	FOR nItemIndex :=1 TO cMAX_VALIDATION_ITEMS DO
		IF eCodeAIType = stCodeInfo.stGS1_Field[nItemIndex].eGS1_AIType THEN
			stItem := stCodeInfo.stGS1_Field[nItemIndex];
			EXIT;
		ELSE
			F_GS1_GetItem := 'Validation Item Not Found';
		END_IF
	END_FOR


	IF stItem.sStartAI <> '' AND stItem.sEndAI <> '' THEN
		nStart := FIND(sFullCode, stItem.sStartAI) + LEN(stItem.sStartAI);
		IF nStart > 0 THEN
			sTemp := RIGHT(sFullCode, LEN(sFullCode) - (nStart - 1));
		ELSE
			sTemp := sFullCode;
		END_IF
		nEnd := FIND(sTemp, stItem.sEndAI);
		IF nEnd = 0 THEN
			nEnd := LEN(sFullCode)+1;
		ELSE
			nEnd := nEnd +(nStart - 1);
		END_IF
	ELSIF stItem.sStartAI <> '' AND stItem.nCodeLength > 0 THEN
		nStart := FIND(sFullCode, stItem.sStartAI) + LEN(stItem.sStartAI);
		nEnd := nStart + stItem.nCodeLength;
	ELSIF stItem.nCodeStartPos > 0 AND stItem.sEndAI <> '' THEN
		nStart := stItem.nCodeStartPos;
		sTemp := RIGHT(sFullCode, LEN(sFullCode) - (nStart - 1));
		nEnd := FIND(sTemp, stItem.sEndAI);
		IF nEnd = 0 THEN
			nEnd := LEN(sFullCode)+1;
		ELSE
			nEnd := nEnd +(nStart - 1);
		END_IF
	ELSIF stItem.nCodeStartPos >= 0 AND stItem.nCodeLength > 0 THEN
		nStart := stItem.nCodeStartPos;
		nEnd := nStart + stItem.nCodeLength;
	ELSE
		nStart := 0;
		nEnd := 0;
	END_IF
	IF nStart > 0 AND nEnd > 0 THEN
		sItem := MID(sFullCode, nEnd - nStart, nStart);
	ELSE
		sItem := '';
	END_IF
ELSE
	sItem := '';
END_IF

F_GS1_GetItem := sItem;

END_FUNCTION

// ---- POUs/METS/Common LIB/08_SOFTWARE LIB/Cog Checker FB/FB_CogCorrection.TcPOU
FUNCTION_BLOCK FB_CogCorrection
VAR_INPUT
	bStart:		BOOL;
	bBailAfterFirstFound: BOOL;
	sSUPI:			STRING[12];
	nCorrectCogID:	INT;
END_VAR
VAR_OUTPUT
	bDone:			BOOL;
	sCorrectSUPI:	ARRAY[1..10] OF STRING[12];
END_VAR
VAR
	sModSUPI:	STRING[12];
	rtrigStart: R_TRIG;
	nChar: INT;
	nPos: INT;
	nStep: INT;
	sChar: STRING[1];
	DIGITS:				STRING[34] :=	'ABCDEFGHJKLMNPQRSTUVWXYZ0123456789';
	nCogResult: INT;
END_VAR

rtrigStart(CLK:= bStart);
IF rtrigStart.Q THEN
	nStep := 1;
END_IF

CASE nStep OF

	1:
		bDone := FALSE;
		MEMSET(ADR(sCorrectSUPI), 0, SIZEOF(sCorrectSUPI));

		sModSUPI := sSUPI;
		nChar := 1;
		nPos := 1;
		nStep := 2;

	2:
		FOR nChar := 1 TO 11 DO
						CheckResult();
			IF bDone THEN
				EXIT;
			END_IF
		END_FOR
		IF NOT(bDone) THEN
			nStep := 3;
		END_IF

	3:
		FOR nChar := 12 TO 23 DO
						CheckResult();
			IF bDone THEN
				EXIT;
			END_IF
		END_FOR
		IF NOT(bDone) THEN
			nStep := 4;
		END_IF


	4:
		FOR nChar := 24 TO 34 DO
						CheckResult();
			IF bDone THEN
				EXIT;
			END_IF
		END_FOR

		IF nPos < 12 THEN
			sModSUPI := sSUPI;
			nPos := nPos+1;
			nStep := 2;
		ELSE
			bDone := TRUE;
			nStep := 0;
		END_IF

END_CASE

ACTION CheckResult:
sChar := MID(DIGITS, 1, nChar);
sModSUPI := REPLACE(sModSUPI, sChar, 1, nPos);
nCogResult := F_COG_Checker(sModSUPI);
IF nCogResult = nCorrectCogID THEN
	MEMMOVE(ADR(sCorrectSUPI[2]), ADR(sCorrectSUPI[1]), SIZEOF(sCorrectSUPI) - SIZEOF(sCorrectSUPI[1]));
	sCorrectSUPI[1] := sModSUPI;
	IF bBailAfterFirstFound THEN
		bDone := TRUE;
		nStep := 0;
	END_IF
END_IF
END_ACTION

END_FUNCTION_BLOCK

// ---- POUs/METS/Common LIB/08_SOFTWARE LIB/Cog Checker FB/F_COG_Checker.TcPOU
FUNCTION F_COG_Checker : INT
VAR_INPUT
	sSUPI		: STRING[12];
END_VAR
VAR
	CogID		: INT;
	biCogID		: T_ULARGE_INTEGER;
	biLenDIGITS	: T_ULARGE_INTEGER;
	biPos		: T_ULARGE_INTEGER;
	biMSUPI_SIZE	: T_ULARGE_INTEGER;
	M			: T_ULARGE_INTEGER;
	biSUPI		: T_ULARGE_INTEGER;
	biPPrime		: T_ULARGE_INTEGER;
	biCODE_SIZE	: T_ULARGE_INTEGER;
	sM			: STRING[255];
	i			: INT;
	Pos			: DINT;
	strSUPI		: STRING[255];
END_VAR
VAR CONSTANT
	CODEGENID_SIZE	: DINT :=	49553;
	CODE_SIZE		: LREAL :=	2386420683693101056;
	DIGITS			: STRING[34] :=	'ABCDEFGHJKLMNPQRSTUVWXYZ0123456789';
	PPrime			: LREAL:= 618222249914457027;
END_VAR

	CogID := -1;
	biCODE_SIZE := LREAL_TO_UINT64(CODE_SIZE);
	biPPrime := LREAL_TO_UINT64(PPrime);

	(*MSUPI_SIZE := 10*366*24*60*1110*8232;*)
	biMSUPI_SIZE := STRING_TO_UINT64('48158385408000');

	bisupi := STRING_TO_UINT64('0');

	FOR i := LEN(sSUPI) TO 1 BY -1 DO
		Pos := FIND(DIGITS, MID(sSUPI, 1, i)) - 1;
		IF Pos >= 0 THEN
			(*supi := (supi* LEN(DIGITS)) + Pos;*)
			biPos.dwLowPart := TO_DWORD(Pos);
			biLenDIGITS.dwLowPart := TO_DWORD(LEN(DIGITS));
			biSUPI := UInt64Mul64(biSUPI, biLenDIGITS);
			biSUPI := UInt64Add64(biSUPI, biPos);
		END_IF
	END_FOR

	strSUPI := UINT64_TO_STRING(biSUPI);
	biPPrime := STRING_TO_UINT64('618222249914457027');
	biCODE_SIZE := STRING_TO_UINT64('2386420683693101056');

	M := F_MulMod(biPPrime, bisupi, biCODE_SIZE);
	sM := UINT64_TO_STRING(M);
	biCogID := UInt64Div64(M, biMSUPI_SIZE);
	CogID := DWORD_TO_INT(biCogID.dwLowPart);

IF CogID <= 0 OR CogID > CODEGENID_SIZE THEN
	CogID := -1;
END_IF

F_COG_Checker := CogID;

END_FUNCTION

// ---- POUs/METS/Common LIB/08_SOFTWARE LIB/Counter FBs/FB_ChangeStateTrig.TcPOU
FUNCTION_BLOCK FB_ChangeStateTrig
(*
Version history:
DATE		|	Version/Author 		|	Remark
----------------------------------------------------------------------------------------------------
16.03.12	|	2.000.001	PSA		|	Original Version.
									|	Monitors a boolean and gives a trigger on change of state
*)
VAR_INPUT
	bInput							: BOOL;			(* Variable to monitor *)
END_VAR
VAR_OUTPUT
	Q								: BOOL;			(* Output trigger *)
END_VAR
VAR
	bLastState						: BOOL;			(* Last known state of the variable *)
	fbTrig							: R_TRIG;		(* Trigger *)
END_VAR

fbTrig(CLK := bInput <> bLastState, Q => Q);
bLastState := bInput;

END_FUNCTION_BLOCK

// ---- POUs/METS/Common LIB/08_SOFTWARE LIB/Counter FBs/FB_CTD32.TcPOU
(* 32-bit counter with count value as VAR_IN_OUT to allow count value to be set externally *)
FUNCTION_BLOCK FB_CTD32
VAR_INPUT
	bInput			: BOOL;		(* FALSE-TRUE increments counter value *)
	bReset			: BOOL;		(* set TRUE to reset counter value to 0 *)
	nThreshold		: UDINT;	(* threshold at which bOutput is set TRUE *)
END_VAR
VAR_IN_OUT
	nCounter		: UDINT;	(* counter value *)
END_VAR
VAR_OUTPUT
	bOutput			: BOOL;		(* nCounter >= nTheshold *)
END_VAR
VAR
	fbInputEdge		: R_TRIG;
END_VAR
(*
-------------------------------------------------------------------------------------------------
Date		Version	Author	Comments
-------------------------------------------------------------------------------------------------
30/01/2015	3.00.00	PB		No change

-------------------------------------------------------------------------------------------------
05/02/10	1.00.00	PB		Initial release

-------------------------------------------------------------------------------------------------
*)

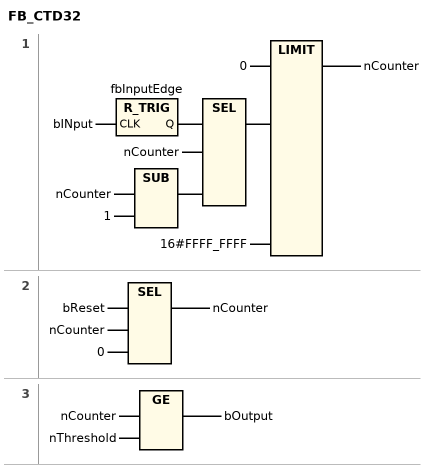
// NETWORK 1
fbInputEdge(CLK := bINput); // R_TRIG
nCounter := LIMIT(0, SEL(fbInputEdge.Q, nCounter, nCounter - 1), 16#FFFF_FFFF);

// NETWORK 2
nCounter := SEL(bReset, nCounter, 0);

// NETWORK 3
bOutput := nCounter >= nThreshold;

END_FUNCTION_BLOCK

// ---- POUs/METS/Common LIB/08_SOFTWARE LIB/Counter FBs/FB_CTU16.TcPOU
(* 16-bit counter with count value as VAR_IN_OUT to allow count value to be set externally *)
FUNCTION_BLOCK FB_CTU16
VAR_INPUT
	bInput			: BOOL;		(* FALSE-TRUE increments counter value *)
	bReset			: BOOL;		(* set TRUE to reset counter value to 0 *)
	nThreshold		: UINT;		(* threshold at which bOutput is set TRUE *)
END_VAR
VAR_IN_OUT
	nCounter		: UINT;		(* counter value *)
END_VAR
VAR_OUTPUT
	bOutput			: BOOL;		(* nCounter >= nTheshold *)
END_VAR
VAR
	fbInputEdge		: R_TRIG;
END_VAR
(*
-------------------------------------------------------------------------------------------------
Date		Version	Author	Comments
-------------------------------------------------------------------------------------------------
30/01/2015	3.00.00	PB		No change

-------------------------------------------------------------------------------------------------
05/02/10	1.00.00	PB		Initial release

-------------------------------------------------------------------------------------------------
*)

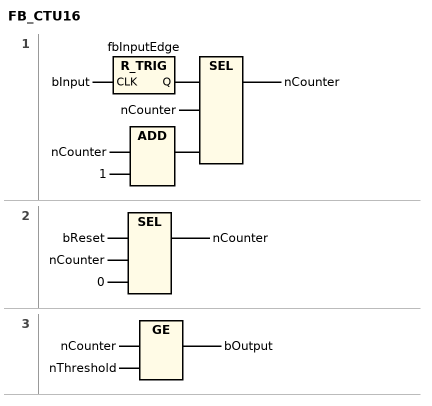
// NETWORK 1
fbInputEdge(CLK := bInput); // R_TRIG
nCounter := SEL(fbInputEdge.Q, nCounter, nCounter + 1);

// NETWORK 2
nCounter := SEL(bReset, nCounter, 0);

// NETWORK 3
bOutput := nCounter >= nThreshold;

END_FUNCTION_BLOCK

// ---- POUs/METS/Common LIB/08_SOFTWARE LIB/Counter FBs/FB_Incrementer.TcPOU
(* pulse incrementer with coarse and fine adjustment *)
FUNCTION_BLOCK FB_Incrementer
VAR_INPUT
	bIncrementHigh		: BOOL;		(* increment fValue in large steps *)
	bIncrementLow		: BOOL;		(* increment fValue in small steps *)
	bDecrementLow		: BOOL;		(* decrement fValue in small steps *)
	bDecrementHigh		: BOOL;		(* decrement fValue in large steps *)
	fLowIncValue		: LREAL;	(* large step change value *)
	fHighIncValue		: LREAL;	(* small step change value *)
END_VAR
VAR_IN_OUT
	fValue				: LREAL;	(* setpoint value *)
END_VAR
VAR
	fbIncrementHigh		: R_TRIG;
	fbIncrementLow		: R_TRIG;
	fbDecrementLow		: R_TRIG;
	fbDecrementHigh		: R_TRIG;
END_VAR
(*
-------------------------------------------------------------------------------------------------
Date		Version	Author	Comments
-------------------------------------------------------------------------------------------------
30/01/2015	3.00.00	PB		No change

-------------------------------------------------------------------------------------------------
26/09/2012	1.09.01	PB		Bug fix - output now LREAL instead of REAL
05/02/10	1.00.00	PB		Initial release

-------------------------------------------------------------------------------------------------
*)

(* add high increment value on rising edge of bIncrementHigh *)
fbIncrementHigh(CLK:= bIncrementHigh);
IF fbIncrementHigh.Q = TRUE THEN

	fValue := fValue + fHighIncValue;
END_IF

(* add low increment value on rising edge of bIncrementLow *)
fbIncrementLow(CLK:= bIncrementLow);
IF fbIncrementLow.Q = TRUE THEN

	fValue := fValue + fLowIncValue;
END_IF

(* subtract low increment value on rising edge of bDecrementLow *)
fbDecrementLow(CLK:= bDecrementLow);
IF fbDecrementLow.Q = TRUE THEN

	fValue := fValue - fLowIncValue;
END_IF

(* subtract high increment value on rising edge of bDecrementHigh *)
fbDecrementHigh(CLK:= bDecrementHigh);
IF fbDecrementHigh.Q = TRUE THEN

	fValue := fValue - fHighIncValue;
END_IF

END_FUNCTION_BLOCK

// ---- POUs/METS/Common LIB/08_SOFTWARE LIB/Counter FBs/FB_InWindow.TcPOU
(* set output when fActPos is within specified window, modulo roll-over is also accounted for *)
FUNCTION_BLOCK FB_InWindow
VAR_INPUT
	bEnable				: BOOL;		(* TRUE = enable output pulse *)
	fStartPos			: LREAL;	(* window start position *)
	fEndPos				: LREAL;	(* window end position *)
	fModuloFactor		: LREAL;	(* axis modulo factor, set to 0 for simple absolute window *)
	fActPos				: LREAL;	(* axis position *)
END_VAR
VAR_OUTPUT
	bInWindow			: BOOL;		(* TRUE = axis modulo position between fStartPos and fEndPos *)
	bStartWindow		: BOOL;		(* TRUE = one-shot pulse when axis has entered position window *)
	bEndWindow			: BOOL;		(* TRUE = one-shot pulse when axis has left position window *)
	fStartPosDiff		: LREAL;	(* pos diff between fStartPos and fActPos when bInWindow was set TRUE *)
END_VAR
VAR
	fbStartWindow		: R_TRIG;
	fbEndWindow			: F_TRIG;
	fCalcStartPos		: LREAL;
	fCalcEndPos			: LREAL;
	fCalcActPos			: LREAL;
END_VAR
(*
-------------------------------------------------------------------------------------------------
Date		Version	Author	Comments
-------------------------------------------------------------------------------------------------
30/01/2015	3.00.00	PB		No change

-------------------------------------------------------------------------------------------------
26/05/2011	1.06.04	PB		Can now set fModuloFactor to 0 to give simple absolute window detection
05/02/10	1.00.00	PB		Initial release

-------------------------------------------------------------------------------------------------

1.	If window is too small and fActPos passes fStartPos AND fEndPos in 1 PLC cycle, bInWindow will NOT be set.
2.	fActPos, fStartPos and fEndPos are automatically corrected for modulo positions, so input values can be
	outside of the modulo window without causing a problem.
*)

(* pulse output enabled *)
IF bEnable = TRUE THEN

	(* use modulo window *)
	IF fModuloFactor > 0 THEN

		(* apply modulo factor to fActPos, fStartPos and fEndPos *)
		fCalcActPos := LMOD(fActPos, fModuloFactor);
		fCalcStartPos := LMOD(fStartPos, fModuloFactor);
		fCalcEndPos := LMOD(fEndPos, fModuloFactor);
	
		(* pulse window does NOT cross modulo position boundary *)
		IF fCalcStartPos <= fCalcEndPos THEN
	
			(* axis modulo position is within defined window *)
			IF fCalcActPos >= fCalcStartPos AND fCalcActPos <= fCalcEndPos THEN
	
				(* set bInWindow output *)
				bInWindow := TRUE;
	
			(* axis modulo position is outside defined window *)
			ELSE
	
				(* reset bInWindow output *)
				bInWindow := FALSE;
			END_IF
	
		(* pulse window DOES cross modulo position boundary *)
		ELSE
	
			(* axis modulo position is within defined window *)
			IF (fCalcActPos >= fCalcStartPos AND fCalcActPos <= fModuloFactor) OR (fCalcActPos >= 0 AND fCalcActPos <= fCalcEndPos) THEN
	
				(* set bInWindow output *)
				bInWindow := TRUE;

			(* axis modulo position is outside defined window *)
			ELSE

				(* reset bInWindow output *)
				bInWindow := FALSE;
			END_IF
		END_IF

	(* use absolute window *)
	ELSE

		(* axis position is within defined window *)
		IF fActPos >= fStartPos AND fActPos <= fEndPos THEN

				(* set bInWindow output *)
			bInWindow := TRUE;

		(* axis position is outside defined window *)
		ELSE

				(* reset bInWindow output *)
			bInWindow := FALSE;
		END_IF
	END_IF


	(* give one-shot output pulse when axis enters defined window *)
	fbStartWindow(
		CLK := bInWindow,
		Q	=> bStartWindow
	);

	(* axis has entered position window *)
	IF bStartWindow = TRUE THEN

		(* calculate difference between target position and actual position when bInWindow is set TRUE *)
		fStartPosDiff := fCalcActPos - fCalcStartPos;
	END_IF

	(* give one-shot output pulse when axis leaves defined window *)
	fbEndWindow(
		CLK := bInWindow,
		Q	=> bEndWindow
	);

(* pulse output enabled *)
ELSE

	(* set outputs to 0, last start window pulse position is not affected *)
	bInWindow := FALSE;
	bStartWindow := FALSE;
	bEndWindow := FALSE;
END_IF

END_FUNCTION_BLOCK

// ---- POUs/METS/Common LIB/08_SOFTWARE LIB/File FBs/FB_FILE_ApendWriteByByte.TcPOU
(* write data from the source array to the target file in byte form *)
FUNCTION_BLOCK FB_FILE_ApendWriteByByte
VAR_INPUT
	bExecute			: BOOL;			(* set TRUE to write file *)
	pSourceAddr			: POINTER TO BYTE;	(* pointer to array of bytes containing data to be written *)
	nSourceSize			: UDINT;		(* number of bytes to write to file *)
	strPathFile			: T_MaxString;	(* path to file to be written *)
	tTimeout			: TIME;			(* timeout *)
END_VAR
VAR_OUTPUT
	bDone				: BOOL;			(* TRUE = file write complete *)
	bBusy				: BOOL;			(* TRUE = file write in progress *)
	bError				: BOOL;			(* TRUE = file write error *)
	nErrorID			: UDINT;		(* error code *)
	nBytesWritten		: UDINT;		(* bytes written to file *)
END_VAR
VAR
	eState				: E_FILE_State;
	eErrorState			: E_FILE_State;
	fbExecute			: R_TRIG;
	pWriteBuffer		: PVOID;
	nWriteBytes			: UDINT;
	fbOpenFile			: FB_FileOpen;
	hTarget				: UINT;
	fbWriteFile			: FB_FileWrite;
	fbCloseFile			: FB_FileClose;
	fbDelay				: TON;
END_VAR
(*
-------------------------------------------------------------------------------------------------
Date		Version	Author	Comments
-------------------------------------------------------------------------------------------------
03/11/2015	3.02.01	PB		Delay after FB_FileClose reduced from 10ms to 2ms
12/08/2015	3.02.00	PB		10ms delay added after FB_FileClose to ensure file has been released by OS before bDone is set TRUE
30/04/2015	3.00.00	PB		Moved from Sewtec_CaseTrace.lib
							Unknown state handling added

-------------------------------------------------------------------------------------------------
21/03/2012	1.37.04	PB		Number of bytes written by FB_FileWrite now checked against nSourceSize, re-write file if valus is incorrect
							Attempt to write file 3 times before returning error
02/03/2010	1.00.00	PB		Initial release

-------------------------------------------------------------------------------------------------
*)

(* rising edge of bExecute *)
fbExecute(CLK := bExecute);

CASE eState OF

	(* idle state *)
	E_FILE_IDLE:

		(* write data to binary file *)
		IF fbExecute.Q = TRUE THEN

			(* reset outputs *)
			bDone := FALSE;
			bBusy := TRUE;
			bError := FALSE;
			nErrorID := 0;
			nBytesWritten := 0;

			(* initialise vars *)
			eErrorState := eState;
			hTarget := 0;
			pWriteBuffer := pSourceAddr;
			nWriteBytes := nSourceSize;

			eState := E_FILE_OPEN;

		(* bExecute has been reset *)
		ELSIF bExecute = FALSE THEN

			bDone := FALSE;
			bBusy := FALSE;
			bError := FALSE;
			nErrorID := 0;

		END_IF


	(* open file *)
	E_FILE_OPEN:

		(* open file for writing in binary mode *)
		fbOpenFile(
			sNetId		:= '',
			sPathName	:= strPathFile,
			nMode		:= FOPEN_MODEAPPEND OR FOPEN_MODEPLUS OR FOPEN_MODEBINARY,
			ePath		:= PATH_GENERIC,
			bExecute	:= TRUE,
			tTimeout	:= tTimeout
		);

		(* file open completed *)
		IF fbOpenFile.bBusy = FALSE THEN

			(* file open completed OK *)
			IF fbOpenFile.bError = FALSE THEN

				(* log file handle for use by subsequent commands *)
				hTarget := fbOpenFile.hFile;

				eState := E_FILE_WRITE;

			(* file open error *)
			ELSE

				(* log error code and failure state *)
				bError := TRUE;
				nErrorID := fbOpenFile.nErrId;
				eErrorState := eState;

				(* abandon attempt to read file *)
				eState := E_FILE_DONE;
			END_IF

			(* close off fbOpenFile *)
			fbOpenFile(bExecute := FALSE);
		END_IF


	(* write file *)
	E_FILE_WRITE:

		(* write data to open file *)
		fbWriteFile(
			sNetId		:= '',
			hFile		:= hTarget,
			pWriteBuff	:= pWriteBuffer,
			cbWriteLen	:= nWriteBytes,
			bExecute	:= TRUE,
			tTimeout	:= tTimeout
		);

		(* file write completed *)
		IF fbWriteFile.bBusy = FALSE THEN

			(* file write completed OK *)
			IF fbWriteFile.bError = FALSE THEN

				(* log total bytes written *)
				nBytesWritten := fbWriteFile.cbWrite;

				eState := E_FILE_CLOSE;

			(* file write error *)
			ELSE

				(* no previous error *)
				IF bError = FALSE THEN

					(* log error code and failure state *)
					bError := TRUE;
					nErrorID := fbWriteFile.nErrId;
					eErrorState := eState;
				END_IF

				eState := E_FILE_CLOSE;
			END_IF

			(* close off fbReadFile *)
			fbWriteFile(bExecute := FALSE);
		END_IF


	(* close file *)
	E_FILE_CLOSE:

		(* close and release file for future use *)
		fbCloseFile(
			sNetId		:= '',
			hFile		:= hTarget,
			bExecute	:= TRUE,
			tTimeout	:= tTimeout,
		);

		(* file close completed *)
		IF fbCloseFile.bBusy = FALSE THEN

			(* file close completed OK *)
			IF fbCloseFile.bError = FALSE THEN

				eState := E_FILE_DONE;

			(* file close error *)
			ELSE

				(* no previous error *)
				IF bError = FALSE THEN

					(* log error code and failure state *)
					bError := TRUE;
					nErrorID := fbCloseFile.nErrId;
					eErrorState := eState;
				END_IF

				eState := E_FILE_DONE;
			END_IF

			(* reset delay timer *)
			fbDelay(IN := FALSE);

			(* close off fbCloseFile *)
			fbCloseFile(bExecute := FALSE);
		END_IF


	(* file access complete *)
	E_FILE_DONE:

		(* file close delay elapsed *)
		IF fbDelay.Q = TRUE THEN

			bDone := TRUE;
			bBusy := FALSE;
	
			eState := E_FILE_IDLE;
		END_IF


(* unknown state*)
ELSE

	eState := E_FILE_IDLE;

	(* update outputs *)
	bDone := TRUE;
	bBusy := FALSE;
	bError := TRUE;
	nErrorID := 16#FFFFFFFF;
	nBytesWritten := 0;
END_CASE

(* delay timer *)
fbDelay(
	IN	:= TRUE,
	PT	:= T#2ms
);

END_FUNCTION_BLOCK

// ---- POUs/METS/Common LIB/08_SOFTWARE LIB/File FBs/FB_FILE_Compare.TcPOU
(* read the attributes of 2 specified files and compare the file sizes in bytes *)
FUNCTION_BLOCK FB_FILE_Compare
VAR_INPUT
	bExecute			: BOOL;			(* set TRUE to compare specified files *)
	strPathFile1		: T_MaxString;	(* full path\file of 1st file for compare *)
	strPathFile2		: T_MaxString;	(* full path\file of 2nd file for compare *)
	tTimeout			: TIME;			(* timeout for each file operation *)
END_VAR
VAR_OUTPUT
	bDone				: BOOL;			(* TRUE = file access complete *)
	bBusy				: BOOL;			(* TRUE = file access in progress *)
	bError				: BOOL;			(* TRUE = error occurred during process *)
	nErrorID			: UDINT;		(* error code *)
	bFileMatchOK		: BOOL;			(* TRUE = files attributes match, valid when bDone = TRUE *)
END_VAR
VAR
	fbExecute			: R_TRIG;
	eState				: E_FILE_State;
	fbReadFileAttrib	: FB_EnumFindFileEntry;
	sFile1Attrib		: ST_FindFileEntry;
	sFile2Attrib		: ST_FindFileEntry;
	eErrorState			: E_FILE_State;
END_VAR
(*
-------------------------------------------------------------------------------------------------
Date		Version	Author	Comments
-------------------------------------------------------------------------------------------------
30/01/2015	3.00.00	PB		Moved from Sewtec_CaseTrace.lib

-------------------------------------------------------------------------------------------------
02/03/2010	1.00.00	PB		Initial release

-------------------------------------------------------------------------------------------------
*)

(* compare files on rising edge of bExecute *)
fbExecute(CLK := bExecute);

CASE eState OF

	(* initialise before scan *)
	E_FILE_IDLE:

		(* start new cycle *)
		IF fbExecute.Q = TRUE THEN

			(* reset outputs *)
			bDone := FALSE;
			bBusy := TRUE;
			bError := FALSE;
			nErrorID := 0;
			eErrorState := eState;
			bFileMatchOK := FALSE;

			eState := E_FILE_READ;

		(* reset status outputs when no cycle is required and bExecute is reset *)
		ELSIF bExecute = FALSE THEN

			bDone := FALSE;
			bBusy := FALSE;
			bError := FALSE;
			nErrorID := 0;
		END_IF


	(* read file 1 *)
	E_FILE_READ:

		(* read file attributes of file 1 *)
		fbReadFileAttrib(
			sNetId		:= '',
			sPathName	:= strPathFile1,
			eCmd		:= eEnumCmd_First,
			bExecute	:= TRUE,
			tTimeout	:= tTimeout,
			stFindFile	=> sFile1Attrib
		);

		(* file attribute read completed *)
		IF fbReadFileAttrib.bBusy = FALSE THEN

			(* file attributes read completed OK *)
			IF fbReadFileAttrib.bError = FALSE THEN

				(* end of entries not found, file exists *)
				IF fbReadFileAttrib.bEOE = FALSE THEN

					(* move to read attributes of File 2 *)
					eState := E_FILE_READ2;

				(* end of entries found, file does not exist *)
				ELSE

					(* no previous error *)
					IF bError = FALSE THEN
	
						bError := TRUE;
						nErrorID := 1;
						eErrorState := eState;
					END_IF

					(* resources held by fbReadFileAttrib released automatically *)
					eState := E_FILE_DONE;
				END_IF

			(* file read error *)
			ELSE

				(* log error code and failure state *)
				bError := TRUE;
				nErrorID := fbReadFileAttrib.nErrID;
				eErrorState := eState;

				(* end of entries found *)
				IF fbReadFileAttrib.bEOE = TRUE THEN

					(* resources released automatically by fbReadFileAttrib, move to compare file details *)
					eState := E_FILE_COMPARE;

				(* end of entries not found *)
				ELSE

					(* release resources held by fbReadFileAttrib *)
					eState := E_FILE_ABORT;
				END_IF
			END_IF

			(* close off fbReadFile *)
			fbReadFileAttrib(bExecute := FALSE);
		END_IF


	(* read file 2 *)
	E_FILE_READ2:

		(* read file attributes of file 2 *)
		fbReadFileAttrib(
			sNetId		:= '',
			sPathName	:= strPathFile2,
			eCmd		:= eEnumCmd_First,
			bExecute	:= TRUE,
			tTimeout	:= tTimeout,
			stFindFile	=> sFile2Attrib
		);

		(* file attribute read completed *)
		IF fbReadFileAttrib.bBusy = FALSE THEN

			(* file attributes read completed OK *)
			IF fbReadFileAttrib.bError = FALSE THEN

				(* end of entries not found, file exists *)
				IF fbReadFileAttrib.bEOE = FALSE THEN

					(* abort fbReadFileAttrib to release resources *)
					eState := E_FILE_ABORT;

				(* end of entries found, file does not exist *)
				ELSE

					(* no previous error *)
					IF bError = FALSE THEN
	
						bError := TRUE;
						nErrorID := 2;
						eErrorState := eState;
					END_IF

					(* resources held by fbReadFileAttrib released automatically *)
					eState := E_FILE_DONE;
				END_IF

			(* file read error *)
			ELSE

				(* log error code and failure state *)
				bError := TRUE;
				nErrorID := fbReadFileAttrib.nErrID;
				eErrorState := eState;

				(* end of entries found *)
				IF fbReadFileAttrib.bEOE = TRUE THEN

					(* resources released automatically by fbReadFileAttrib, move to compare file details *)
					eState := E_FILE_COMPARE;

				(* end of entries not found *)
				ELSE

					(* release resources held by fbReadFileAttrib *)
					eState := E_FILE_ABORT;
				END_IF
			END_IF

			(* close off fbReadFile *)
			fbReadFileAttrib(bExecute := FALSE);
		END_IF


	(* abort fbReadFileAttrib to release all resources *)
	E_FILE_ABORT:

		(* abort fbReadFileAttrib to release internal resources *)
		fbReadFileAttrib(
			eCmd		:= eEnumCmd_Abort,
			bExecute	:= TRUE,
		);

		(* abort file attricute read complete *)
		IF fbReadFileAttrib.bBusy = FALSE THEN

			(* abort file attricute read completed OK *)
			IF fbReadFileAttrib.bError = FALSE THEN

				(* no error occurred during file attribute read sequences *)
				IF bError = FALSE THEN

					(* move to COMPARE file attributes state *)
					eState := E_FILE_COMPARE;

				(* error occurred during file attribute read sequences *)
				ELSE

					(* move to COMPARE file attributes state *)
					eState := E_FILE_DONE;
				END_IF

			(* abort error *)
			ELSE

				(* no error occurred in previous states *)
				IF bError = FALSE THEN

					(* log error code and failure state *)
					bError := TRUE;
					nErrorID := fbReadFileAttrib.nErrID;
					eErrorState := eState;
				END_IF

				eState := E_FILE_DONE;
			END_IF

			(* close off fbReadFileAttrib *)
			fbReadFileAttrib(bExecute := FALSE);
		END_IF


	(* compare file attributes *)
	E_FILE_COMPARE:

		(* check if file size values (high and low dwords) are equal *)
		IF sFile1Attrib.fileSize.dwLowPart = sFile2Attrib.fileSize.dwLowPart
			AND sFile1Attrib.fileSize.dwHighPart = sFile2Attrib.fileSize.dwHighPart THEN

			bFileMatchOK := TRUE;	(* file sizes identical *)
		END_IF

		(* compare done *)
		eState := E_FILE_DONE;


	(* file access complete *)
	E_FILE_DONE:

		bDone := TRUE;
		bBusy := FALSE;

		(* return to IDLE state *)
		eState := E_FILE_IDLE;
END_CASE

END_FUNCTION_BLOCK

// ---- POUs/METS/Common LIB/08_SOFTWARE LIB/File FBs/FB_FILE_Copy.TcPOU
(* copy file(s) from SOURCE folder to TARGET folder, wildcard chars '*' and '?' can be used *)
FUNCTION_BLOCK FB_FILE_Copy
VAR_INPUT
	bExecute			: BOOL;			(* set TRUE to copy multiple files *)
	strPathSource		: T_MaxString;	(* folder path for SOURCE file*)
	strPathTarget		: T_MaxString;	(* folder path for TARGET file *)
	strFileName			: T_MaxString;	(* name of file to be copied *)
	tTimeout			: TIME;			(* timeout for each file operation *)
END_VAR
VAR_OUTPUT
	bDone				: BOOL;			(* TRUE = file access complete *)
	bBusy				: BOOL;			(* TRUE = file access in progress *)
	bError				: BOOL;			(* TRUE = error occurred during process *)
	nErrorID			: UDINT;		(* error code *)
	strOutputFile		: T_MaxString;	(* name of file that failed *)
END_VAR
VAR
	fbExecute			: R_TRIG;
	eState				: E_FILE_State;
	eErrorState			: E_FILE_State;
	fbFindFile			: FB_EnumFindFileEntry;
	eCommand			: E_EnumCmdType;
	strFoundFile		: T_MaxString;
	fbCopyFile			: FB_FILE_CopyByByte;
END_VAR
(*
-------------------------------------------------------------------------------------------------
Date		Version	Author	Comments
-------------------------------------------------------------------------------------------------
30/01/2015	3.00.00	PB		Moved from Sewtec_CaseTrace.lib

-------------------------------------------------------------------------------------------------
27/09/2010	1.05.03	PB		If a file cannot be copied, FB will now continue to next file in list rather than just abort and report an error
							strOutputFile will contain the name of the last file that failed
22/03/2010	1.02.00	PB		Initial release

-------------------------------------------------------------------------------------------------
*)

(* compare files on rising edge of bExecute *)
fbExecute(CLK := bExecute);

CASE eState OF

	(* idle state *)
	E_FILE_IDLE:

		(* start new cycle *)
		IF fbExecute.Q = TRUE THEN

			(* reset outputs *)
			bDone := FALSE;
			bBusy := TRUE;
			bError := FALSE;
			nErrorID := 0;
			strOutputFile := '';
			eErrorState := eState;

			eCommand := eEnumCmd_First;

			eState := E_FILE_FINDFILE;

		(* reset status outputs when no cycle is required and bExecute is reset *)
		ELSIF bExecute = FALSE THEN

			bDone := FALSE;
			bBusy := FALSE;
			bError := FALSE;
			nErrorID := 0;
			strOutputFile := '';
		END_IF


	(* find file *)
	E_FILE_FINDFILE:

		(* get file name *)
		fbFindFile(
			sNetId		:= '',
			sPathName	:= CONCAT(strPathSource, strFileName),
			eCmd		:= eCommand,
			bExecute	:= TRUE,
			tTimeout	:= T#1s,
		);

		(* get file name complete *)
		IF fbFindFile.bBusy = FALSE THEN

			(* get file name completed OK *)
			IF fbFindFile.bError = FALSE THEN

				(* file found *)
				IF fbFindFile.bEOE = FALSE THEN

					eCommand := eEnumCmd_Next;

					(* ignore filenames '.' and '..' *)
					IF fbFindFile.stFindFile.sFileName <> '.' AND fbFindFile.stFindFile.sFileName <> '..' THEN

						strFoundFile := fbFindFile.stFindFile.sFileName;
						eState := E_FILE_COPY;
					END_IF

				(* end of file list *)
				ELSE

					(* copy files complete *)
					eState := E_FILE_DONE;
				END_IF

			(* get file name error *)
			ELSE

				(* no error has previously occurred *)
				IF bError = FALSE THEN

					(* log error code and failure state *)
					bError := TRUE;
					nErrorID := fbFindFile.nErrId;
					eErrorState := eState;
				END_IF

				(* abandon attempt to copy files *)
				eState := E_FILE_ABORT;
			END_IF

			(* close off fbFindFile *)
			fbFindFile(bExecute := FALSE);
		END_IF


	(* copy file to TARGET folder *)
	E_FILE_COPY:

		(* copy files *)
		fbCopyFile(
			bExecute		:= TRUE,
			strPathSource	:= strPathSource,
			strPathTarget	:= strPathTarget,
			strFileName		:= strFoundFile,
			tTimeout		:= tTimeout,
		);

		(* copy file complete *)
		IF fbCopyFile.bDone = TRUE THEN

			(* copy file completed OK *)
			IF fbCopyFile.bError = FALSE THEN

				eState := E_FILE_FINDFILE;

			(* copy file error *)
			ELSE

				(* no error has previously occurred *)
				IF bError = FALSE THEN

					(* log error code and failure state *)
					strOutputFile := CONCAT(strPathSource, strFoundFile);
					bError := TRUE;
					nErrorID := fbCopyFile.nErrorID;
					eErrorState := eState;
				END_IF

				eState := E_FILE_FINDFILE;
			END_IF

			(* close off fbCopyFile *)
			fbCopyFile(bExecute := FALSE);
		END_IF


	(* abort file entry list *)
	E_FILE_ABORT:

		(* abort file entry list *)
		fbFindFile(
			sNetId		:= '',
			sPathName	:= '',
			eCmd		:= eEnumCmd_Abort,
			bExecute	:= TRUE,
			tTimeout	:= T#1s,
		);

		(* abort file entry complete *)
		IF fbFindFile.bBusy = FALSE THEN

			(* abort file entry completed OK *)
			IF fbFindFile.bError = FALSE THEN

				eState := E_FILE_DONE;

			(* abort file entry error *)
			ELSE

				(* no error has previously occurred *)
				IF bError = FALSE THEN

					(* log error code and failure state *)
					bError := TRUE;
					nErrorID := fbFindFile.nErrId;
					eErrorState := eState;
				END_IF

				(* abandon attempt to copy files *)
				eState := E_FILE_DONE;
			END_IF

			(* close off fbFindFile *)
			fbFindFile(bExecute := FALSE);
		END_IF


	(* file access complete *)
	E_FILE_DONE:

		bDone := TRUE;
		bBusy := FALSE;

		(* return to IDLE state *)
		eState := E_FILE_IDLE;

END_CASE

END_FUNCTION_BLOCK

// ---- POUs/METS/Common LIB/08_SOFTWARE LIB/File FBs/FB_FILE_CopyByByte.TcPOU
(* copy file from SOURCE to TARGET and verify, wildcard chars NOT allowed *)
FUNCTION_BLOCK FB_FILE_CopyByByte
VAR_INPUT
	bExecute			: BOOL;			(* set TRUE to copy file *)
	strPathSource		: T_MaxString;	(* folder path for SOURCE file*)
	strPathTarget		: T_MaxString;	(* folder path for TARGET file *)
	strFileName			: T_MaxString;	(* name of file to be copied*)
	tTimeout			: TIME;			(* timeout for each file operation *)
END_VAR
VAR_OUTPUT
	bDone				: BOOL;			(* TRUE = file access complete *)
	bBusy				: BOOL;			(* TRUE = file access in progress *)
	bError				: BOOL;			(* TRUE = error occurred during process *)
	nErrorID			: UDINT;		(* error code *)
END_VAR
VAR
	fbExecute			: R_TRIG;
	eState				: E_FILE_State;
	eErrorState			: E_FILE_State;
	fbGetFileSize		: FB_FILE_GetFileInfo;
	bFileSizeNotZero	: BOOL;
	fbOpenFile			: FB_FileOpen;
	hFileHandleSource	: UINT;
	hFileHandleTarget	: UINT;
	fbReadFile			: FB_FileRead;
	arrFileBytes		: ARRAY[0..32767] OF BYTE;
	nBytesRead			: UDINT;
	fbWriteFile			: FB_FileWrite;
	fbCloseFile			: FB_FileClose;
	fbFileCompare		: FB_FILE_Compare;
	bEOF				: BOOL;
END_VAR
(*
-------------------------------------------------------------------------------------------------
Date		Version	Author	Comments
-------------------------------------------------------------------------------------------------
30/01/2015	3.00.00	PB		Moved from Sewtec_CaseTrace.lib

-------------------------------------------------------------------------------------------------
23/03/2010	1.02.00	PB		strFileName input added
							Source and target files split into source/target path and filename inputs
02/03/2010	1.00.00	PB		Initial release

-------------------------------------------------------------------------------------------------
*)

(* compare files on rising edge of bExecute *)
fbExecute(CLK := bExecute);

CASE eState OF

	(* initialise before scan *)
	E_FILE_IDLE:

		(* start new cycle *)
		IF fbExecute.Q = TRUE THEN

			(* reset outputs *)
			bDone := FALSE;
			bBusy := TRUE;
			bError := FALSE;
			nErrorID := 0;
			eErrorState := eState;

			eState := E_FILE_GETSIZE;

		(* reset status outputs when no cycle is required and bExecute is reset *)
		ELSIF bExecute = FALSE THEN

			bDone := FALSE;
			bBusy := FALSE;
			bError := FALSE;
			nErrorID := 0;
		END_IF


	(* check source file size *)
	E_FILE_GETSIZE:

		(* get source file info *)
		fbGetFileSize(
			bExecute		:= TRUE,
			strPathSource	:= strPathSource,
			strFileName		:= strFileName,
			tTimeout		:= tTimeout,
		);

		(* read file size complete *)
		IF fbGetFileSize.bDone = TRUE THEN

			(* read file size completed OK *)
			IF fbGetFileSize.bError = FALSE THEN

				(* file size > 0 bytes *)
				IF fbGetFileSize.nFileSizeLo > 0 OR fbGetFileSize.nFileSizeHi > 0 THEN

					bFileSizeNotZero := TRUE;

				(* file size = 0 bytes *)
				ELSE

					bFileSizeNotZero := FALSE;
				END_IF

				eState := E_FILE_OPEN;

			(* read file size error *)
			ELSE

				eErrorState := eState;
				eState := E_FILE_DONE;
			END_IF

			fbGetFileSize(bExecute := FALSE);
		END_IF


	(* open source file *)
	E_FILE_OPEN:

		(* if source file size > 0 bytes, open for reading in binary mode *)
		fbOpenFile(
			sNetId		:= '',
			sPathName	:= CONCAT(strPathSource, strFileName),
			nMode		:= FOPEN_MODEREAD OR FOPEN_MODEBINARY,
			ePath		:= PATH_GENERIC,
			bExecute	:= bFileSizeNotZero,
			tTimeout	:= tTimeout,
			hFile		=> hFileHandleSource
		);

		(* source file open completed *)
		IF fbOpenFile.bBusy = FALSE THEN

			(* source file open completed OK *)
			IF fbOpenFile.bError = FALSE THEN

				eState := E_FILE_OPEN2;

			(* file open error *)
			ELSE

				(* no error has previously occurred *)
				IF bError = FALSE THEN

					(* log error code and failure state *)
					bError := TRUE;
					nErrorID := fbOpenFile.nErrId;
					eErrorState := eState;
				END_IF

				(* abandon attempt to read file *)
				eState := E_FILE_DONE;
			END_IF

			(* close off fbOpenSourceFile *)
			fbOpenFile(bExecute := FALSE);
		END_IF


	(* open destination file *)
	E_FILE_OPEN2:

		(* open specified file for reading in binary mode *)
		fbOpenFile(
			sNetId		:= '',
			sPathName	:= CONCAT(strPathTarget, strFileName),
			nMode		:= FOPEN_MODEWRITE OR FOPEN_MODEBINARY,
			ePath		:= PATH_GENERIC,
			bExecute	:= TRUE,
			tTimeout	:= tTimeout,
			hFile		=> hFileHandleTarget
		);

		(* destination file open completed *)
		IF fbOpenFile.bBusy = FALSE THEN

			(* destination file open completed OK *)
			IF fbOpenFile.bError = FALSE THEN

				eState := E_FILE_READ;

			(* file open error *)
			ELSE

				(* no error has previously occurred *)
				IF bError = FALSE THEN

					(* log error code and failure state *)
					bError := TRUE;
					nErrorID := fbOpenFile.nErrId;
					eErrorState := eState;
				END_IF

				(* close destination file *)
				eState := E_FILE_CLOSE2;
			END_IF

			(* close off fbOpenFile *)
			fbOpenFile(bExecute := FALSE);
		END_IF



	(* read source file *)
	E_FILE_READ:

		(* if source file size > 0 bytes, read data in file *)
		fbReadFile(
			sNetId		:= '',
			hFile		:= hFileHandleSource,
			pReadBuff	:= ADR(arrFileBytes),
			cbReadLen	:= SIZEOF(arrFileBytes),
			bExecute	:= bFileSizeNotZero,
			tTimeout	:= tTimeout
		);

		(* file read completed *)
		IF fbReadFile.bBusy = FALSE THEN

			(* file read completed OK *)
			IF fbReadFile.bError = FALSE THEN

				bEOF := fbReadFile.bEOF;
				nBytesRead := fbReadFile.cbRead;

				(* end of file not reached *)
				IF bEOF = FALSE THEN

					(* more data to be copied *)
					eState := E_FILE_WRITE;

				(* end of file reached *)
				ELSE

					(* all data copied, close files *)
					eState := E_FILE_CLOSE;
				END_IF

			(* file read error *)
			ELSE

				(* no error has previously occurred *)
				IF bError = FALSE THEN

					(* log error code and failure state *)
					bError := TRUE;
					nErrorID := fbReadFile.nErrId;
					eErrorState := eState;
				END_IF

				(* abandon read and close file *)
				eState := E_FILE_CLOSE;
			END_IF

			(* close off fbReadFile *)
			fbReadFile(bExecute := FALSE);
		END_IF


	(* write data to target file *)
	E_FILE_WRITE:

		(* write data to file *)
		fbWriteFile(
			sNetId		:= '',
			hFile		:= hFileHandleTarget,
			pWriteBuff	:= ADR(arrFileBytes),
			cbWriteLen	:= nBytesRead,
			bExecute	:= TRUE,
			tTimeout	:= tTimeout
		);

		(* file write completed *)
		IF fbWriteFile.bBusy = FALSE THEN

			(* file write completed OK *)
			IF fbWriteFile.bError = FALSE THEN

				(* end of file or filesize is 0 bytes*)
				IF bEOF = TRUE OR bFileSizeNotZero = FALSE THEN

					(* close files *)
					eState := E_FILE_CLOSE;

				(* more data to read *)
				ELSE

					eState := E_FILE_READ;
				END_IF

			(* file read error *)
			ELSE

				(* no error has previously occurred *)
				IF bError = FALSE THEN

					(* log error code and failure state *)
					bError := TRUE;
					nErrorID := fbWriteFile.nErrId;
					eErrorState := eState;
				END_IF

				(* abandon read and close file *)
				eState := E_FILE_CLOSE;
			END_IF

			(* close off fbWriteFile *)
			fbWriteFile(bExecute := FALSE);
		END_IF


	(* close destination file *)
	E_FILE_CLOSE:

		(* close destination file *)
		fbCloseFile(
			sNetId		:= '',
			hFile		:= hFileHandleTarget,
			bExecute	:= TRUE,
			tTimeout	:= tTimeout,
		);

		(* file close completed *)
		IF fbCloseFile.bBusy = FALSE THEN

			(* file close completed OK *)
			IF fbCloseFile.bError = FALSE THEN

				(* close source file *)
				eState := E_FILE_CLOSE2;

			(* file close error *)
			ELSE

				(* no error occurred with FileOpen or FileRead *)
				IF bError = FALSE THEN

					(* log error code and failure state *)
					bError := TRUE;
					nErrorID := fbCloseFile.nErrId;
					eErrorState := eState;
				END_IF

				(* close source file *)
				eState := E_FILE_CLOSE2;
			END_IF

			(* close off fbCloseFile *)
			fbCloseFile(bExecute := FALSE);
		END_IF


	(* close source file *)
	E_FILE_CLOSE2:

		(* if source file size > 0 bytes, it would have been opened so must be closed *)
		fbCloseFile(
			sNetId		:= '',
			hFile		:= hFileHandleSource,
			bExecute	:= bFileSizeNotZero,
			tTimeout	:= tTimeout,
		);

		(* file close completed *)
		IF fbCloseFile.bBusy = FALSE THEN

			(* file close completed OK *)
			IF fbCloseFile.bError = FALSE THEN

				(* no error has occurred *)
				IF bError = FALSE THEN

					(* compare source and destination files *)
					eState := E_FILE_COMPARE;

				(* error has occurred *)
				ELSE

					(* file copy complete *)
					eState := E_FILE_DONE;
				END_IF

			(* file close error *)
			ELSE

				(* no error occurred with FileOpen or FileRead *)
				IF bError = FALSE THEN

					(* log error code and failure state *)
					bError := TRUE;
					nErrorID := fbCloseFile.nErrId;
					eErrorState := eState;
				END_IF

				(* go to DONE state *)
				eState := E_FILE_DONE;
			END_IF

			(* close off fbCloseFile *)
			fbCloseFile(bExecute := FALSE);
		END_IF


	(* compare files *)
	E_FILE_COMPARE:

		(* compare source and target files to ensure copy was successful *)
		fbFileCompare(
			bExecute		:= TRUE,
			strPathFile1	:= CONCAT(strPathSource, strFileName),
			strPathFile2	:= CONCAT(strPathTarget, strFileName),
			tTimeout		:= T#1s,
		);

		(* file compare completed *)
		IF fbFileCompare.bBusy = FALSE THEN

			(* file compare completed OK *)
			IF fbFileCompare.bError = FALSE THEN

				eState := E_FILE_DONE;

			(* file read error *)
			ELSE

				(* no error has previously occurred *)
				IF bError = FALSE THEN

					(* log error code and failure state *)
					bError := TRUE;
					nErrorID := fbFileCompare.nErrorID;
					eErrorState := eState;
				END_IF

				(* sequence complete *)
				eState := E_FILE_DONE;
			END_IF

			(* close off fbFileCompare *)
			fbFileCompare(bExecute := FALSE);
		END_IF


	(* file access complete *)
	E_FILE_DONE:

		bDone := TRUE;
		bBusy := FALSE;

		(* return to IDLE state *)
		eState := E_FILE_IDLE;

END_CASE

END_FUNCTION_BLOCK

// ---- POUs/METS/Common LIB/08_SOFTWARE LIB/File FBs/FB_FILE_GetFileInfo.TcPOU
(* check if a file exists by attempting to read the file attributes *)
FUNCTION_BLOCK FB_FILE_GetFileInfo
VAR_INPUT
	bExecute			: BOOL;			(* set TRUE to get file info *)
	strPathSource		: T_MaxString;	(* folder path for SOURCE file, wildcard chars '*' and '?' can be used *)
	strFileName		: T_MaxString;	(* name of file to be copied, wildcard chars '*' and '?' can be used *)
	tTimeout			: TIME;			(* timeout for each file operation *)
END_VAR
VAR_OUTPUT
	bDone			: BOOL;			(* TRUE = file access complete *)
	bBusy			: BOOL;			(* TRUE = file access in progress *)
	bError			: BOOL;			(* TRUE = error occurred during process *)
	nErrorID			: UDINT;		(* error code *)
	bFileExists		: BOOL;			(* TRUE = specified file exists *)
	bFileSizeNotZero	: BOOL;			(* TRUE = file size >0 bytes *)
	bFileNotFound		: BOOL;			(* TRUE = specified file not found *)
	nFileSizeLo		: UDINT;		(* file size low part (<4Gb) *)
	nFileSizeHi		: UDINT;		(* file size high part (>4Gb) *)
	strFileFound		: T_MaxString;	(* full name of file found *)
END_VAR
VAR
	fbExecute			: R_TRIG;
	eState			: E_FILE_State;
	eErrorState		: E_FILE_State;
	fbReadFileAttrib	: FB_EnumFindFileEntry;
END_VAR

(* compare files on rising edge of bExecute *)
fbExecute(CLK := bExecute);

CASE eState OF

	(* initialise before scan *)
	E_FILE_IDLE:

		(* start new cycle *)
		IF fbExecute.Q = TRUE THEN

			(* reset outputs *)
			bDone := FALSE;
			bBusy := TRUE;
			bError := FALSE;
			nErrorID := 0;
			eErrorState := eState;
			bFileExists := FALSE;
			bFileSizeNotZero := FALSE;
			bFileNotFound := FALSE;
			nFileSizeLo := 0;
			nFileSizeHi := 0;
			strFileFound := '';

			eState := E_FILE_READ;

		(* reset status outputs when no cycle is required and bExecute is reset *)
		ELSIF bExecute = FALSE THEN

			bDone := FALSE;
			bBusy := FALSE;
			bError := FALSE;
			nErrorID := 0;
			bFileExists := FALSE;
			bFileSizeNotZero := FALSE;
			bFileNotFound := FALSE;
			nFileSizeLo := 0;
			nFileSizeHi := 0;
			strFileFound := '';
		END_IF


	(* read file *)
	E_FILE_READ:

		(* read file attributes of file *)
		fbReadFileAttrib(
			sNetId		:= '',
			sPathName	:= CONCAT(strPathSource, strFileName),
			eCmd		:= eEnumCmd_First,
			bExecute	:= TRUE,
			tTimeout	:= tTimeout
		);

		(* file read completed *)
		IF fbReadFileAttrib.bBusy = FALSE THEN

			(* file read completed OK *)
			IF fbReadFileAttrib.bError = FALSE THEN

				(* file was found *)
				IF fbReadFileAttrib.bEOE = FALSE THEN

					(* update outputs *)
					bFileExists := TRUE;
					nFileSizeLo := fbReadFileAttrib.stFindFile.fileSize.dwLowPart;
					nFileSizeHi := fbReadFileAttrib.stFindFile.fileSize.dwHighPart;
					strFileFound := fbReadFileAttrib.stFindFile.sFileName;

					(* file size > 0 bytes *)
					IF nFileSizeLo > 0 OR nFileSizeHi > 0 THEN

						bFileSizeNotZero := TRUE;
					END_IF

					(* release internal resources *)
					eState := E_FILE_ABORT;

				(* file was not found *)
				ELSE

					(* internal resources released automatically, no need to abort *)
					bFileNotFound := TRUE;
					eState := E_FILE_DONE;
				END_IF

			(* file read error *)
			ELSE

				(* no previous error *)
				IF bError = FALSE THEN

					(* log error code and failure state *)
					bError := TRUE;
					nErrorID := fbReadFileAttrib.nErrID;
					eErrorState := eState;
				END_IF

				(* abort to release resources *)
				eState := E_FILE_ABORT;
			END_IF

			(* close off fbReadFileAttrib *)
			fbReadFileAttrib(bExecute := FALSE);
		END_IF


	(* abort fbReadFileAttrib to release all resources *)
	E_FILE_ABORT:

		(* abort fbReadFileAttrib to release internal resources *)
		fbReadFileAttrib(
			eCmd		:= eEnumCmd_Abort,
			bExecute	:= TRUE
		);

		(* abort file attricute read complete *)
		IF fbReadFileAttrib.bBusy = FALSE THEN

			(* abort file attricute read completed OK *)
			IF fbReadFileAttrib.bError = FALSE THEN

				(* move to COMPARE file attributes state *)
				eState := E_FILE_DONE;

			(* abort error *)
			ELSE

				(* no error occurred in previous states *)
				IF bError = FALSE THEN

					(* log error code and failure state *)
					bError := TRUE;
					nErrorID := fbReadFileAttrib.nErrID;
					eErrorState := eState;
				END_IF

				eState := E_FILE_DONE;
			END_IF

			(* close off fbReadFileAttrib *)
			fbReadFileAttrib(bExecute := FALSE);
		END_IF


	(* file access complete *)
	E_FILE_DONE:

		bDone := TRUE;
		bBusy := FALSE;

		(* return to IDLE state *)
		eState := E_FILE_IDLE;
END_CASE

END_FUNCTION_BLOCK

// ---- POUs/METS/Common LIB/08_SOFTWARE LIB/File FBs/FB_FILE_Delete.TcPOU
(* delete files from SOURCE folder, wildcard chars '*' and '?' can be used *)
FUNCTION_BLOCK FB_FILE_Delete
VAR_INPUT
	bExecute			: BOOL;			(* set TRUE to copy multiple files *)
	strPathSource		: T_MaxString;	(* folder path for SOURCE file, must NOT contain file name *)
	strFileName			: T_MaxString;	(* name of file to be copied *)
	tTimeout			: TIME;			(* timeout for each file operation *)
END_VAR
VAR_OUTPUT
	bDone				: BOOL;			(* TRUE = file access complete *)
	bBusy				: BOOL;			(* TRUE = file access in progress *)
	bError				: BOOL;			(* TRUE = error occurred during process *)
	nErrorID			: UDINT;		(* error code *)
	strOutputFile		: T_MaxString;	(* name of file that failed *)
END_VAR
VAR
	fbExecute			: R_TRIG;
	eState				: E_FILE_State;
	eErrorState			: E_FILE_State;
	fbGetFileName		: FB_EnumFindFileEntry;
	eCommand			: E_EnumCmdType;
	strFoundFile		: T_MaxString;
	fbDeleteFile		: FB_FileDelete;
END_VAR
(*
-------------------------------------------------------------------------------------------------
Date		Version	Author	Comments
-------------------------------------------------------------------------------------------------
30/01/2015	3.00.00	PB		Moved from Sewtec_CaseTrace.lib

-------------------------------------------------------------------------------------------------
27/09/2010	1.05.03	PB		If a file cannot be deleted, FB will now continue to next file in list rather than just abort and report an error
							strOutputFile will contain the name of the last file that failed
22/03/2010	1.02.00	PB		Name changed from FB_FILE_PurgeDirectory to FB_FILE_DeleteFiles
							Bug with deleting all files using '*.*' fixed
							Source file split into path and filename inputs
19/03/2010	1.01.00	PB		Initial release

-------------------------------------------------------------------------------------------------
*)

(* compare files on rising edge of bExecute *)
fbExecute(CLK := bExecute);

CASE eState OF

	(* idle state *)
	E_FILE_IDLE:

		(* start new cycle *)
		IF fbExecute.Q = TRUE THEN

			(* reset outputs *)
			bDone := FALSE;
			bBusy := TRUE;
			bError := FALSE;
			nErrorID := 0;
			strOutputFile := '';
			eErrorState := eState;

			eCommand := eEnumCmd_First;

			eState := E_FILE_CHECKIFEXISTS;

		(* reset status outputs when no cycle is required and bExecute is reset *)
		ELSIF bExecute = FALSE THEN

			bDone := FALSE;
			bBusy := FALSE;
			bError := FALSE;
			nErrorID := 0;
			strOutputFile := '';
		END_IF


	(* find file *)
	E_FILE_CHECKIFEXISTS:

		(* get file name *)
		fbGetFileName(
			sNetId		:= '',
			sPathName	:= CONCAT(strPathSource, strFileName),
			eCmd		:= eCommand,
			bExecute	:= TRUE,
			tTimeout	:= tTimeout,
		);

		(* get file name complete *)
		IF fbGetFileName.bBusy = FALSE THEN

			(* get file name completed OK *)
			IF fbGetFileName.bError = FALSE THEN

				(* file found *)
				IF fbGetFileName.bEOE = FALSE THEN

					eCommand := eEnumCmd_Next;

					(* ignore filenames '.' and '..' *)
					IF fbGetFileName.stFindFile.sFileName <> '.' AND fbGetFileName.stFindFile.sFileName <> '..' THEN

						strFoundFile := fbGetFileName.stFindFile.sFileName;
						eState := E_FILE_DELETE;
					END_IF

				(* end of file list *)
				ELSE

					(* copy files complete *)
					eState := E_FILE_DONE;
				END_IF

			(* get file name error *)
			ELSE

				(* no error has previously occurred *)
				IF bError = FALSE THEN

					(* log error code and failure state *)
					bError := TRUE;
					nErrorID := fbGetFileName.nErrId;
					eErrorState := eState;
				END_IF

				(* abandon attempt to copy files *)
				eState := E_FILE_ABORT;
			END_IF

			(* close off fbGetFileName *)
			fbGetFileName(bExecute := FALSE);
		END_IF


	(* delete file from SOURCE folder *)
	E_FILE_DELETE:

		(* delete files *)
		fbDeleteFile(
			sNetId		:= '',
			sPathName	:= CONCAT(strPathSource, strFoundFile),
			ePath		:= PATH_GENERIC,
			bExecute	:= TRUE,
			tTimeout	:= tTimeout
		);

		(* delete file complete *)
		IF fbDeleteFile.bBusy = FALSE THEN

			(* delete file completed OK *)
			IF fbDeleteFile.bError = FALSE THEN

				eState := E_FILE_CHECKIFEXISTS;

			(* copy file error *)
			ELSE

				(* no error has previously occurred *)
				IF bError = FALSE THEN

					(* log error code and failure state *)
					strOutputFile := fbDeleteFile.sPathName;
					bError := TRUE;
					nErrorID := fbDeleteFile.nErrId;
					eErrorState := eState;
				END_IF

				(*eState := E_FILE_ABORT;*)
				eState := E_FILE_CHECKIFEXISTS;
			END_IF

			(* close off fbDeleteFile *)
			fbDeleteFile(bExecute := FALSE);
		END_IF


	(* abort file entry list *)
	E_FILE_ABORT:

		(* abort file entry list *)
		fbGetFileName(
			sNetId		:= '',
			sPathName	:= '',
			eCmd		:= eEnumCmd_Abort,
			bExecute	:= TRUE,
			tTimeout	:= tTimeout,
		);

		(* abort file entry complete *)
		IF fbGetFileName.bBusy = FALSE THEN

			(* abort file entry completed OK *)
			IF fbGetFileName.bError = FALSE THEN

				eState := E_FILE_DONE;

			(* abort file entry error *)
			ELSE

				(* no error has previously occurred *)
				IF bError = FALSE THEN

					(* log error code and failure state *)
					bError := TRUE;
					nErrorID := fbGetFileName.nErrId;
					eErrorState := eState;
				END_IF

				(* abandon attempt to copy files *)
				eState := E_FILE_DONE;
			END_IF

			(* close off fbGetFileName *)
			fbGetFileName(bExecute := FALSE);
		END_IF


	(* file access complete *)
	E_FILE_DONE:

		bDone := TRUE;
		bBusy := FALSE;

		(* return to IDLE state *)
		eState := E_FILE_IDLE;

END_CASE

END_FUNCTION_BLOCK

// ---- POUs/METS/Common LIB/08_SOFTWARE LIB/File FBs/FB_FILE_DeleteOldFiles.TcPOU
(* keeps a folder clear of files by deleting files older than a specified period and deleting oldest files to keep number of files to the max specified level *)
FUNCTION_BLOCK FB_FILE_DeleteOldFiles
VAR_INPUT
	bExecute			: BOOL;			(* set TRUE to clear old or excess files from a directory *)
	nMaxFiles			: UINT;			(* max files allowed in directory *)
	strPath				: T_MaxString;	(* folder path *)
	strFile				: T_MaxString;	(* file name, '*' and '?' wildcard chars are supported *)
	tMaxFileAge			: TIME;			(* max file age, older files will be deleted *)
END_VAR
VAR_OUTPUT
	bDone				: BOOL;			(* TRUE = delete old files complete *)
	bBusy				: BOOL;			(* TRUE = delete old files in progress *)
	bError				: BOOL;			(* TRUE = delete old files error *)
	nErrorID			: UDINT;		(* error code *)
	nFilesFound			: UINT;			(* total files found in folder *)
	nFilesDeleted		: UINT;			(* total files deleted from folder *)
END_VAR
VAR
	eState				: E_FILE_DeleteOldFilesState;
	eErrorState			: E_FILE_DeleteOldFilesState;
	fbExecute			: R_TRIG;
	strPathInternal		: T_MaxString;
	strFileInternal		: T_MaxString;
	fbGetSystemTime		: GETSYSTEMTIME;
	nMaxFileAge			: T_ULARGE_INTEGER;
	nCurrentDateTime	: T_ULARGE_INTEGER;
	fbFindFile			: FB_EnumFindFileEntry;
	nCurrentFile		: UINT;
	nFileCreationTime	: T_ULARGE_INTEGER;
	arrFileTime			: ARRAY[1..1000] OF T_ULARGE_INTEGER;
	nIndex				: UINT;
	nMaxIndex			: UINT;
	nFileTimeThreshold	: T_ULARGE_INTEGER;
	fbDeleteFile		: FB_FileDelete;
	strFileName			: T_MaxString;
END_VAR
(*
-------------------------------------------------------------------------------------------------
DATE		Version	Author	Comments
-------------------------------------------------------------------------------------------------
30/01/2015	3.00.00	PB		Moved from Sewtec_CaseTrace.lib

-------------------------------------------------------------------------------------------------
03/08/2012	1.39.00	PB		Bug fix - correct files now deleted if file creation date order does not follow alphabetical name order
26/03/2012	1.38.00	PB		Initial release

-------------------------------------------------------------------------------------------------
*)

(* rising edge of bExecute *)
fbExecute(CLK:= bExecute);

CASE eState OF

	(* Idle *)
	E_OLDFILE_IDLE:

		(* rising edge of bExecute *)
		IF fbExecute.Q = TRUE THEN

			nMaxIndex := UDINT_TO_UINT(SIZEOF(arrFileTime) / SIZEOF(arrFileTime[1]));
			strPathInternal := strPath;
			strFileInternal := strFile;

			(* clear file creation time array *)
			MEMSET(ADR(arrFileTime), 16#00, SIZEOF(arrFileTime));

			bDone := FALSE;
			bBusy := TRUE;
			bError := FALSE;
			nErrorID := 0;
			nFilesFound := 0;
			nFilesDeleted := 0;
			nCurrentFile := 0;

			eErrorState := eState;

			(* get system time as UTC for local computer *)
			fbGetSystemTime(
				timeLoDW	=> nCurrentDateTime.dwLowPart,
				timeHiDW	=> nCurrentDateTime.dwHighPart
			);

			(* convert TIME (1 = 1ms) to T_ULARGE_INTEGER (1 = 100ns) *)
			nMaxFileAge := UInt32x32To64(TIME_TO_UDINT(tMaxFileAge), 10000);

			eState := E_OLDFILE_FILELIST1;

		(* no action, bExecute has been reset to FALSE *)
		ELSIF bExecute = FALSE THEN

			bDone := FALSE;
			bBusy := FALSE;
			bError := FALSE;
			nErrorID := 0;
			nFilesFound := 0;
			nFilesDeleted := 0;
		END_IF


	(* build and sort list of file creation times *)
	E_OLDFILE_FILELIST1:

		(* find next file *)
		fbFindFile(
			sNetId		:= '',
			sPathName	:= CONCAT(strPathInternal, strFileInternal),
			eCmd		:= SEL(nCurrentFile = 0, eEnumCmd_Next, eEnumCmd_First),
			bExecute	:= TRUE,
			tTimeout	:= T#1s,
		);

		(* find file complete *)
		IF fbFindFile.bBusy = FALSE THEN

			(* find file completed OK *)
			IF fbFindFile.bError = FALSE THEN

				(* end of list not reached *)
				IF fbFindFile.bEOE = FALSE THEN

					(* another file found *)
					nCurrentFile := nCurrentFile + 1;
					nFilesFound := nCurrentFile;
					nFileCreationTime := F_FileTimeToULarge(fbFindFile.stFindFile.creationTime);

					(* file list is sorted newest file (largest time-stamp value) at nIndex = 1 *)
					(* file time is newer than 1st file in list *)
					IF UInt64Cmp64(nFileCreationTime, arrFileTime[1]) = 1 THEN

						(* shift existing  file times up by 1 index *)
						MEMMOVE(ADR(arrFileTime[2]), ADR(arrFileTime[1]), SIZEOF(arrFileTime) - SIZEOF(arrFileTime[1]));

						(* add new file time to array *)
						arrFileTime[1] := nFileCreationTime;

					(* file time is same age or older than 1st file in list *)
					ELSE

						(* scan list of file creation times *)
						FOR nIndex := 1 TO nCurrentFile DO

							(* insertion point found *)
							IF (UInt64Cmp64(nFileCreationTime, arrFileTime[nIndex]) = -1 OR UInt64Cmp64(nFileCreationTime, arrFileTime[nIndex]) = 0) AND UInt64Cmp64(nFileCreationTime, arrFileTime[nIndex + 1]) = 1 THEN

								(* shift older file times up by 1 index *)
								MEMMOVE(ADR(arrFileTime[nIndex + 2]), ADR(arrFileTime[nIndex + 1]), SIZEOF(arrFileTime[1]) * (nMaxIndex - nIndex - 1));

								(* add new file time to array *)
								arrFileTime[nIndex + 1] := nFileCreationTime;

								(* finish scan as insertion point has been found *)
								EXIT;
							END_IF
						END_FOR
					END_IF

				(* end of list *)
				ELSE

					(* no of files in folder exceeds max limit *)
					IF nFilesFound > nMaxFiles THEN

						(* calculate file time threshold *)
						nFileTimeThreshold := arrFileTime[nMaxFiles];

					(* no of files in folder OK *)
					ELSE

						(* calculate file time threshold *)
						nFileTimeThreshold := UInt64Sub64(nCurrentDateTime, nMaxFileAge);
					END_IF

					(* restart new file list *)
					nCurrentFile := 0;

					eState := E_OLDFILE_FILELIST2;
				END_IF

			(* find file error *)
			ELSE

				IF bError = FALSE THEN

					bError := TRUE;
					eErrorState := eState;
					nErrorID := fbFindFile.nErrID;
				END_IF

				eState := E_OLDFILE_ABORTFILELIST;
			END_IF

			(* close off fbFindFile *)
			fbFindFile(bExecute := FALSE);
		END_IF


	(* find file and check creation date to see if it should be deleted *)
	E_OLDFILE_FILELIST2:

		(* find next file *)
		fbFindFile(
			sNetId		:= '',
			sPathName	:= CONCAT(strPathInternal, strFileInternal),
			eCmd		:= SEL(nCurrentFile = 0, eEnumCmd_Next, eEnumCmd_First),
			bExecute	:= TRUE,
			tTimeout	:= T#1s,
		);

		(* find file complete *)
		IF fbFindFile.bBusy = FALSE THEN

			(* fbFindFile file completed OK *)
			IF fbFindFile.bError = FALSE THEN

				(* end of list not reached *)
				IF fbFindFile.bEOE = FALSE THEN

					nCurrentFile := nCurrentFile + 1;
					nFileCreationTime := F_FileTimeToULarge(fbFindFile.stFindFile.creationTime);

					(* nFileCreationTime <= file time threshold *)
					IF UInt64Cmp64(nFileCreationTime, nFileTimeThreshold) = -1 OR UInt64Cmp64(nFileCreationTime, nFileTimeThreshold) = 0 THEN

						(* name of file to be deleted *)
						strFileName := fbFindFile.stFindFile.sFileName;

						eState := E_OLDFILE_DELETEFILELIST2;
					END_IF

				(* end of list *)
				ELSE

					eState := E_OLDFILE_DONE;
				END_IF

			(* find file error *)
			ELSE

				IF bError = FALSE THEN

					bError := TRUE;
					eErrorState := eState;
					nErrorID := fbFindFile.nErrID;
				END_IF

				eState := E_OLDFILE_ABORTFILELIST;
			END_IF

			(* close off fbFindFile *)
			fbFindFile(bExecute := FALSE);
		END_IF


	(* delete file *)
	E_OLDFILE_DELETEFILELIST2:

		(* delete file *)
		fbDeleteFile(
			sNetId		:= '',
			sPathName	:= CONCAT(strPathInternal, strFileName),
			ePath		:= PATH_GENERIC,
			bExecute	:= TRUE,
			tTimeout	:= T#1s,
		);

		(* delete file complete *)
		IF fbDeleteFile.bBusy = FALSE THEN

			(* file delete completed OK *)
			IF fbDeleteFile.bError = FALSE THEN

				nFilesDeleted := nFilesDeleted + 1;
			END_IF

			eState := E_OLDFILE_FILELIST2;

			(* close off fbDeleteFile *)
			fbDeleteFile(bExecute := FALSE);
		END_IF


	E_OLDFILE_ABORTFILELIST:

		(* find next file *)
		fbFindFile(
			sNetId		:= '',
			sPathName	:= CONCAT(strPath, strFile),
			eCmd		:= eEnumCmd_Abort,
			bExecute	:= TRUE,
			tTimeout	:= T#1s,
		);

		(* find file complete *)
		IF fbFindFile.bBusy = FALSE THEN

			eState:= E_OLDFILE_DONE;

			fbFindFile(bExecute := FALSE);
		END_IF


	(* complete *)
	E_OLDFILE_DONE:

		bDone := TRUE;
		bBusy := FALSE;

		eState := E_OLDFILE_IDLE;


	(* unknown state *)
	ELSE

		eState := E_OLDFILE_IDLE;

END_CASE

END_FUNCTION_BLOCK

// ---- POUs/METS/Common LIB/08_SOFTWARE LIB/Maths FBs/F_FileTimeToULarge.TcPOU
(* convert value from 64-bit T_FILETIME to 64-bit T_ULARGE_INTEGER *)
FUNCTION F_FileTimeToULarge : T_ULARGE_INTEGER
VAR_INPUT
	sFileTime		: T_FILETIME;
END_VAR
VAR
END_VAR
(*
-------------------------------------------------------------------------------------------------
Date		Version	Author	Comments
-------------------------------------------------------------------------------------------------
30/01/2015	3.00.00	PB		Moved from Sewtec_CaseTrace.lib

-------------------------------------------------------------------------------------------------
26/03/2012	1.38.00	PB		Initial release

-------------------------------------------------------------------------------------------------
*)

MEMMOVE(ADR(F_FileTimeToULarge), ADR(sFileTime), SIZEOF(F_FileTimeToULarge));

END_FUNCTION

// ---- POUs/METS/Common LIB/08_SOFTWARE LIB/File FBs/FB_FILE_GetFileList.TcPOU
(* build list of files and associated attributes, wildcard chars can be used *)
FUNCTION_BLOCK FB_FILE_GetFileList
VAR_INPUT
	bExecute			: BOOL;			(* set TRUE to build file list *)
	strPath				: T_MaxString;	(* folder path *)
	strFile				: T_MaxString;	(* fil name, wild card chars '*' and '?' can be used *)
	pFileList			: POINTER TO ST_FindFileEntry;		(* pointer to file list, ARRAY[1..xx] OF ST_FindFileEntry *)
	nFileListSize		: UDINT;		(* file list size in bytes *)
	tTimeout			: TIME;			(* timeout *)
END_VAR
VAR_OUTPUT
	bDone				: BOOL;			(* TRUE = file list complete *)
	bBusy				: BOOL;			(* TRUE = file list in progress *)
	bError				: BOOL;			(* TRUE = file list error *)
	nErrorID			: UDINT;		(* error code *)
	nFilesFound			: UDINT;		(* number of files found *)
END_VAR
VAR
	fbExecute			: R_TRIG;
	eState				: E_FILE_State;
	eErrorState			: E_FILE_State;
	pPointer			: POINTER TO ST_FindFileEntry;
	nPointer			: PVOID;

	strPathFile			: T_MaxString;
	fbGetFileList		: FB_EnumFindFileList;
	sFile				: ST_FindFileEntry;
	nMaxFiles			: UDINT;
END_VAR
(*
-------------------------------------------------------------------------------------------------
Date		Version	Author	Comments
-------------------------------------------------------------------------------------------------
30/01/2015	3.00.00	PB		Moved from Sewtec_CaseTrace.lib

-------------------------------------------------------------------------------------------------
21/03/2012	1.37.04	PB		Abort file list if fbGetFileList returns an error
							Pointer handling to file array changed and simplified
02/08/2011	1.27.01	PB		Bug fix - file list was not cleared if no files were found
							Bug fix - 1st file found is now placed at start of file list
14/06/2011	1.20.00	PB		Initial release

-------------------------------------------------------------------------------------------------
*)

(* build file list on risign edge of bExecute *)
fbExecute(CLK := bExecute);

CASE eState OF

	(* IDLE state *)
	E_FILE_IDLE:

		(* build file list *)
		IF fbExecute.Q = TRUE THEN

			(* initialise variables *)
			pPointer := pFileList;
			nMaxFiles := nFileListSize / SIZEOF(sFile);
			nFilesFound := 0;
			strPathFile := CONCAT(strPath, strFile);

			eState := E_FILE_FINDFILE;

		(* no action requird *)
		ELSIF bExecute= FALSE THEN

			bDone := FALSE;
			bBusy := FALSE;
			bError := FALSE;
			nErrorID := 0;
		END_IF


	(* build file list *)
	E_FILE_FINDFILE:

		(* get file list *)
		fbGetFileList(
			sNetId		:= '',
			sPathName	:= strPathFile,
			eCmd		:= eEnumCmd_First,
			pFindList	:= ADR(sFile),
			cbFindList	:= SIZEOF(sFile),
			bExecute	:= TRUE,
			tTimeout	:= tTimeout
		);

		(* get file list complete *)
		IF fbGetFileList.bBusy = FALSE THEN

			(* get file list completed OK *)
			IF fbGetFileList.bError = FALSE THEN

				(* 1 or more files found *)
				IF fbGetFileList.bEOE = FALSE THEN

					(* move new file info into 1st location in file list *)
					MEMMOVE(pPointer, ADR(sFile), SIZEOF(sFile));
					nFilesFound := 1;

					(* calculate pointer to next value in file list array *)
					nPointer := pPointer;					(* convert pointer to UDINT *)
					nPointer := nPointer + SIZEOF(sFile);	(* add offset *)
					pPointer := nPointer;					(* convert UDINT back to pointer *)

					eState := E_FILE_NEXTFILE;

				(* no files found *)
				ELSE

					(* move new file info into file list *)
					MEMSET(pFileList, 16#00, nFileListSize);
					nFilesFound := 0;

					eState := E_FILE_DONE;
				END_IF

			(* file list error *)
			ELSE

				(* no previous error has occurred *)
				IF bError = FALSE THEN

					bError := TRUE;
					nErrorID := fbGetFileList.nErrID;
					eErrorState := eState;
				END_IF

				eState := E_FILE_CLOSELIST;
			END_IF

			(* close off fbGetFileList *)
			fbGetFileList(bExecute := FALSE);
		END_IF


	(* next file *)
	E_FILE_NEXTFILE:

		(* get next file in list *)
		fbGetFileList(
			sNetId		:= '',
			sPathName	:= strPathFile,
			eCmd		:= eEnumCmd_Next,
			pFindList	:= ADR(sFile),
			cbFindList	:= SIZEOF(sFile),
			bExecute	:= TRUE,
			tTimeout	:= tTimeout
		);

		(* get next file complete *)
		IF fbGetFileList.bBusy = FALSE THEN

			(* get next file completed OK *)
			IF fbGetFileList.bError = FALSE THEN

				(* end of file list has been reached *)
				IF fbGetFileList.bEOE = TRUE THEN

					(* space still available in file list buffer *)
					IF nFilesFound < nMaxFiles THEN

						(* clear unused locations in buffer *)
						MEMSET(pPointer, 16#00, SIZEOF(sFile) * (nMaxFiles - nFilesFound));
					END_IF

					(* file list completed and closed automatically *)
					eState := E_FILE_DONE;

				(* add file to list *)
				ELSE

					(* space available in file list buffer *)
					IF nFilesFound <= nMaxFiles THEN

						(* move file info to file list array *)
						MEMMOVE(pPointer, ADR(sFile), SIZEOF(sFile));

						(* calculate pointer to next value in file list array *)
						nPointer := pPointer;					(* convert pointer to UDINT *)
						nPointer := nPointer + SIZEOF(sFile);	(* add offset *)
						pPointer := nPointer;					(* convert UDINT back to pointer *)
					END_IF

					(* increment number of files found *)
					nFilesFound := nFilesFound + fbGetFileList.nFindFiles;
				END_IF

			(* get next file error *)
			ELSE

				(* no previous error *)
				IF bError = FALSE THEN

					bError := TRUE;
					nErrorID := fbGetFileList.nErrID;
					eErrorState := eState;
				END_IF

				eState := E_FILE_CLOSELIST;
			END_IF

			(* close off fbGetFileList *)
			fbGetFileList(bExecute := FALSE);
		END_IF


	(* close file list *)
	E_FILE_CLOSELIST:

		(* abort file list *)
		fbGetFileList(
			sNetId		:= '',
			eCmd		:= eEnumCmd_Abort,
			bExecute	:= TRUE,
			tTimeout	:= tTimeout
		);

		(* file list close complete *)
		IF fbGetFileList.bBusy = FALSE THEN

			(* file list close completed OK *)
			IF fbGetFileList.bError = FALSE THEN

				eState := E_FILE_DONE;

			(* file list close error *)
			ELSE

				(* no previous error *)
				IF bError = FALSE THEN

					bError := TRUE;
					nErrorID := fbGetFileList.nErrID;
					eErrorState := eState;
				END_IF

				eState := E_FILE_DONE;
			END_IF

			(* close off fbGetFileList *)
			fbGetFileList(bExecute := FALSE);
		END_IF


	(* done *)
	E_FILE_DONE:

		bDone := TRUE;
		bBusy := FALSE;

		eState := E_FILE_IDLE;

END_CASE

END_FUNCTION_BLOCK

// ---- POUs/METS/Common LIB/08_SOFTWARE LIB/File FBs/FB_FILE_MoveWithDate.TcPOU
(* move file(s) from SOURCE folder to TARGET folder, wildcard chars '*' and '?' can be used *)
FUNCTION_BLOCK FB_FILE_MoveWithDate
VAR_INPUT
	bExecute			: BOOL;			(* set TRUE to copy multiple files *)
	strPathSource		: T_MaxString;	(* path of SOURCE folder *)
	strPathTarget		: T_MaxString;	(* path of TARGET folder *)
	strFileName		: T_PCM_Filename;	(* file name to be moved, wildcard chars ('*', '?') can be used *)
	stCTDateTime		: ST_SYSTEM_DateTime;	(* CaseTrace date/time structure *)
	tTimeout			: TIME;			(* timeout for each file operation *)
END_VAR
VAR_OUTPUT
	bDone			: BOOL;			(* TRUE = file access complete *)
	bBusy			: BOOL;			(* TRUE = file access in progress *)
	bError			: BOOL;			(* TRUE = error occurred during process *)
	nErrorID			: UDINT;		(* error code *)
	strOutputFile		: T_PCM_Filename;	(* name of file that failed *)
	strLastFileMoved		: T_MaxString;
END_VAR
VAR
	fbExecute			: R_TRIG;
	eState			: E_FILE_State;
	eErrorState		: E_FILE_State;
	fbFindFile			: FB_EnumFindFileEntry;
	eCommand		: E_EnumCmdType;
	strDateToFile		: STRING(8);
	strTimeToFile		: STRING(6);
	strTimeStamp		: STRING(16);
	strNewFileName	: T_PCM_Filename;
	strFoundFile		: T_PCM_Filename;
	fbDeleteFile		: FB_FileDelete;
	fbMoveFile		: FB_FileRename;
END_VAR
(*
-------------------------------------------------------------------------------------------------
Date		Version	Author	Comments
-------------------------------------------------------------------------------------------------
30/01/2015	3.00.00	PB		Moved from Sewtec_CaseTrace.lib

-------------------------------------------------------------------------------------------------
27/09/2010	1.05.03	PB		If a file cannot be moved, FB will now continue to next file in list rather than just abort and report an error
							strOutputFile will contain the name of the last file that failed
23/03/2010	1.02.00	PB		Name changed from FB_FILE_MoveByByte to FB_FILE_Move
							Internal operation changed to delete target file (if exists) and move source file to target file using FB_FileRename
							Support for wildcard chars added to allow multiple files to be moved
02/03/2010	1.00.00	PB		Initial release

-------------------------------------------------------------------------------------------------
*)

(* compare files on rising edge of bExecute *)
fbExecute(CLK := bExecute);

CASE eState OF

	(* idle state *)
	E_FILE_IDLE:

		(* start new cycle *)
		IF fbExecute.Q = TRUE THEN

			(* reset outputs *)
			bDone := FALSE;
			bBusy := TRUE;
			bError := FALSE;
			nErrorID := 0;
			strOutputFile := '';
			strLastFileMoved :='';
			eErrorState := eState;

			(* start new file list *)
			eCommand := eEnumCmd_First;


			strDateToFile := F_StringWildcard('#YYYYMMDD#', stCTDateTime.sSystemTime);
			strTimeToFile:= F_StringWildcard('#hhmmss#', stCTDateTime.sSystemTime);
			strTimeStamp := F_CONCAT3(strDateToFile, '_' , strTimeToFile);

			eState := E_FILE_FINDFILE;

		(* reset status outputs when no cycle is required and bExecute is reset *)
		ELSIF bExecute = FALSE THEN

			bDone := FALSE;
			bBusy := FALSE;
			bError := FALSE;
			nErrorID := 0;
			strOutputFile := '';
		END_IF


	(* find file *)
	E_FILE_FINDFILE:

		(* get file name *)
		fbFindFile(
			sNetId		:= '',
			sPathName	:= CONCAT(strPathSource, strFileName),
			eCmd		:= eCommand,
			bExecute	:= TRUE,
			tTimeout	:= T#1s,
		);

		(* find file complete *)
		IF fbFindFile.bBusy = FALSE THEN

			(* find file completed OK *)
			IF fbFindFile.bError = FALSE THEN

				(* file found *)
				IF fbFindFile.bEOE = FALSE THEN

					(* find next file in list *)
					eCommand := eEnumCmd_Next;

					(* ignore filenames '.' and '..' *)
					IF fbFindFile.stFindFile.sFileName <> '.' AND fbFindFile.stFindFile.sFileName <> '..' THEN

						strFoundFile := fbFindFile.stFindFile.sFileName;
						strNewFileName := F_FILE_AppendStringToFileName( strFoundFile, strTimeStamp, '.xml');
						eState := E_FILE_DELETE;
					END_IF

				(* end of file list *)
				ELSE

					(* copy files complete *)
					eState := E_FILE_DONE;
				END_IF

			(* find file error *)
			ELSE

				(* no error has previously occurred *)
				IF bError = FALSE THEN

					(* log error code and failure state *)
					bError := TRUE;
					nErrorID := fbFindFile.nErrId;
					eErrorState := eState;
				END_IF

				(* abandon attempt to copy files *)
				eState := E_FILE_ABORT;
			END_IF

			(* close off fbFindFile *)
			fbFindFile(bExecute := FALSE);
		END_IF


	(* delete target file *)
	E_FILE_DELETE:

		(* delete file *)
		fbDeleteFile(
			sNetId		:= '',
			sPathName	:= CONCAT(strPathTarget, strNewFileName),
			ePath		:= PATH_GENERIC,
			bExecute	:= TRUE,
			tTimeout	:= tTimeout
		);

		(* file delete completed *)
		IF fbDeleteFile.bBusy = FALSE THEN

			(* file delete completed OK *)
			IF fbDeleteFile.bError = FALSE THEN

				eState := E_FILE_MOVE;

			(* file delete error *)
			ELSE

				(* file did not exist, OK to move file to TARGET folder *)
				IF fbDeleteFile.nErrId = 1804 THEN

					eState := E_FILE_MOVE;

				(* other file delete error occurred *)
				ELSE

					(* no error has previously occurred *)
					IF bError = FALSE THEN

						(* log error code and failure state *)
						strOutputFile := fbDeleteFile.sPathName;
						bError := TRUE;
						nErrorID := fbDeleteFile.nErrId;
						eErrorState := eState;
					END_IF

					(* move on to next file *)
					eState := E_FILE_FINDFILE;
				END_IF

			END_IF

			(* close off fbFileDelete *)
			fbDeleteFile(bExecute := FALSE);
		END_IF


	(* move source file to destination file *)
	E_FILE_MOVE:

		(* move file *)
		fbMoveFile(
			sNetId		:= '',
			sOldName	:= CONCAT(strPathSource, strFoundFile),
			sNewName	:= CONCAT(strPathTarget, strNewFileName),
			ePath		:= PATH_GENERIC,
			bExecute	:= TRUE,
			tTimeout	:= tTimeout,
		);
		
		(* file move completed *)
		IF fbMoveFile.bBusy = FALSE THEN

			(* file move completed OK *)
			IF fbMoveFile.bError = FALSE THEN

				strLastFileMoved :=strFoundFile;

			(* file move error *)
			ELSE

				(* no error has previously occurred *)
				IF bError = FALSE THEN

					(* log error code and failure state *)
					strOutputFile := fbMoveFile.sOldName;
					bError := TRUE;
					nErrorID := fbMoveFile.nErrId;
					eErrorState := eState;
				END_IF
			END_IF

			(* move on to next file *)
			eState := E_FILE_FINDFILE;

			(* close off fbMoveFile *)
			fbMoveFile(bExecute := FALSE);
		END_IF


	(* abort file entry list *)
	E_FILE_ABORT:

		(* abort file entry list *)
		fbFindFile(
			sNetId		:= '',
			sPathName	:= '',
			eCmd		:= eEnumCmd_Abort,
			bExecute	:= TRUE,
			tTimeout	:= T#1s,
		);

		(* abort file entry complete *)
		IF fbFindFile.bBusy = FALSE THEN

			(* abort file entry completed OK *)
			IF fbFindFile.bError = FALSE THEN

				eState := E_FILE_DONE;

			(* abort file entry error *)
			ELSE

				(* no error has previously occurred *)
				IF bError = FALSE THEN

					(* log error code and failure state *)
					bError := TRUE;
					nErrorID := fbFindFile.nErrId;
					eErrorState := eState;
				END_IF

				(* abandon attempt to copy files *)
				eState := E_FILE_DONE;
			END_IF

			(* close off fbFindFile *)
			fbFindFile(bExecute := FALSE);
		END_IF


	(* file access complete *)
	E_FILE_DONE:

		bDone := TRUE;
		bBusy := FALSE;

		(* return to IDLE state *)
		eState := E_FILE_IDLE;

END_CASE

END_FUNCTION_BLOCK

// ---- POUs/METS/Common LIB/08_SOFTWARE LIB/File FBs/F_FILE_AppendStringToFileName.TcPOU
FUNCTION F_FILE_AppendStringToFileName : T_MaxString

VAR_INPUT
	sFilename 						: T_MaxString;
	sExtraString					: T_MaxString;
	sExtension 					: T_FileExtension;
END_VAR
VAR
	sResult 							: T_MaxString;
	nDotPosition						: INT;
END_VAR

F_FILE_AppendStringToFileName :='';

IF LEFT(sExtension,1) <> cDOT_CHAR THEN (*No leading dot character found, so add it *)
	sExtension := CONCAT(cDOT_CHAR, sExtension);
END_IF

nDotPosition := FIND(sFilename, sExtension);

IF nDotPosition <> 0 THEN
	sResult := LEFT(sFilename, nDotPosition-1);
	sResult := F_CONCAT4(sResult, '_',sExtraString,sExtension);
ELSE
	sResult := '';
END_IF

F_FILE_AppendStringToFileName := sResult;

END_FUNCTION

// ---- POUs/METS/Common LIB/08_SOFTWARE LIB/File FBs/FB_FILE_ReadByByte.TcPOU
(* read data from specified by in source file to the target array in byte form *)
FUNCTION_BLOCK FB_FILE_ReadByByte
VAR_INPUT
	bExecute			: BOOL;			(* set TRUE to read file *)
	pTargetAddr			: POINTER TO BYTE;	(* pointer to array of bytes where data from file will be stored *)
	nTargetSize			: UDINT;		(* size of data array assigned to received data from file *)
	nByteOffset			: DINT;			(* offset to 1st byte of file to be loaded *)
	strPathFile			: T_MaxString;	(* full path\file of input file *)
	tTimeout			: TIME;			(* timeout for each file operation *)
END_VAR
VAR_OUTPUT
	bDone				: BOOL;			(* TRUE = file access complete *)
	bBusy				: BOOL;			(* TRUE = file access in progress *)
	bError				: BOOL;			(* TRUE = error occurred during process *)
	nErrorID			: UDINT;		(* error code *)
	bEOF				: BOOL;			(* TRUE = end of file found *)
	nBytesRead			: UDINT;		(* number of bytes read from specified file *)
END_VAR
VAR
	eState				: E_FILE_State;
	eErrorState			: E_FILE_State;
	fbExecute			: R_TRIG;
	fbOpenFile			: FB_FileOpen;
	hFileHandle			: UINT;
	fbSetTargetByte		: FB_FileSeek;
	fbReadFile			: FB_FileRead;
	fbCloseFile			: FB_FileClose;
END_VAR
(*
-------------------------------------------------------------------------------------------------
Date		Version	Author	Comments
-------------------------------------------------------------------------------------------------
30/01/2015	3.00.00	PB		Moved from Sewtec_CaseTrace.lib

-------------------------------------------------------------------------------------------------
23/03/2010	1.01.00	PB		nByteOffset input added to specify 1st byte of file to be loaded
02/03/2010	1.00.00	PB		Initial release

-------------------------------------------------------------------------------------------------
*)

(* load XML file on rising edge of bExecute *)
fbExecute(CLK := bExecute);

CASE eState OF

	(* initialise before scan *)
	E_FILE_IDLE:

		(* start new cycle *)
		IF fbExecute.Q = TRUE THEN

			(* reset outputs *)
			bDone := FALSE;
			bBusy := TRUE;
			bError := FALSE;
			nErrorID := 0;
			eErrorState := eState;

			eState := E_FILE_OPEN;

		(* reset status outputs when no cycle is required and bExecute is reset *)
		ELSIF bExecute = FALSE THEN

			bDone := FALSE;
			bBusy := FALSE;
			bError := FALSE;
			nErrorID := 0;
			bEOF := FALSE;
			nBytesRead := 0;
		END_IF


	(* open file *)
	E_FILE_OPEN:

		(* open specified file for reading in binary mode *)
		fbOpenFile(
			sNetId		:= '',
			sPathName	:= strPathFile,
			nMode		:= FOPEN_MODEREAD OR FOPEN_MODEBINARY,
			ePath		:= PATH_GENERIC,
			bExecute	:= TRUE,
			tTimeout	:= tTimeout,
			hFile		=> hFileHandle
		);

		(* file open completed *)
		IF fbOpenFile.bBusy = FALSE THEN

			(* file open completed OK *)
			IF fbOpenFile.bError = FALSE THEN

				nBytesRead := 0;
				eState := E_FILE_SEEK;

			(* file open error *)
			ELSE

				(* no error occurred with FileOpen or FileRead *)
				IF bError = FALSE THEN

					(* log error code and failure state *)
					bError := TRUE;
					nErrorID := fbOpenFile.nErrId;
					eErrorState := eState;
				END_IF

				(* abandon attempt to read file *)
				eState := E_FILE_DONE;
			END_IF

			(* close off fbOpenFile *)
			fbOpenFile(bExecute := FALSE);
		END_IF


	(* set 1st byte to be read from file *)
	E_FILE_SEEK:

		(* initialise file pointer *)
		fbSetTargetByte(
			sNetId	:= '',
			hFile	:= hFileHandle,
			nSeekPos:= nByteOffset,
			eOrigin	:= SEEK_SET,
			bExecute:= TRUE,
			tTimeout:= tTimeout
		);

		(* initialise pointer complete *)
		IF fbSetTargetByte.bBusy = FALSE THEN

			(* initialise pointer completed OK *)
			IF fbSetTargetByte.bError = FALSE THEN

				eState := E_FILE_READ;


			(* pointer could not be initialised *)
			ELSE

				(* no previous error occurred *)
				IF bError = FALSE THEN

					(* log error code and failure state *)
					bError := TRUE;
					nErrorID := fbSetTargetByte.nErrId;
					eErrorState := eState;
				END_IF

				(* abandon read and close file *)
				eState := E_FILE_CLOSE;
			END_IF

			(* close off fbSetTargetByte *)
			fbSetTargetByte(bExecute := FALSE);
		END_IF


	(* read file *)
	E_FILE_READ:

		(* read data in from open file *)
		fbReadFile(
			sNetId		:= '',
			hFile		:= hFileHandle,
			pReadBuff	:= pTargetAddr,
			cbReadLen	:= nTargetSize,
			bExecute	:= TRUE,
			tTimeout	:= tTimeout,
			cbRead		=> nBytesRead,
			bEOF		=> bEOF
		);

		(* file read completed *)
		IF fbReadFile.bBusy = FALSE THEN

			(* file read completed OK *)
			IF fbReadFile.bError = FALSE THEN

				eState := E_FILE_CLOSE;

			(* file read error *)
			ELSE

				(* no error occurred with FileOpen or FileRead *)
				IF bError = FALSE THEN

					(* log error code and failure state *)
					bError := TRUE;
					nErrorID := fbReadFile.nErrId;
					eErrorState := eState;
				END_IF

				(* abandon read and close file *)
				eState := E_FILE_CLOSE;
			END_IF

			(* close off fbReadFile *)
			fbReadFile(bExecute := FALSE);
		END_IF


	(* close file *)
	E_FILE_CLOSE:

		(* close and release file for future use *)
		fbCloseFile(
			sNetId		:= '',
			hFile		:= hFileHandle,
			bExecute	:= TRUE,
			tTimeout	:= tTimeout,
		);

		(* file close completed *)
		IF fbCloseFile.bBusy = FALSE THEN

			(* file close completed OK *)
			IF fbCloseFile.bError = FALSE THEN

				(* go to DONE state *)
				eState := E_FILE_DONE;

			(* file close error *)
			ELSE

				(* no error occurred with FileOpen or FileRead *)
				IF bError = FALSE THEN

					(* log error code and failure state *)
					bError := TRUE;
					nErrorID := fbCloseFile.nErrId;
					eErrorState := eState;
				END_IF

				(* go to DONE state *)
				eState := E_FILE_DONE;
			END_IF

			(* close off fbCloseFile *)
			fbCloseFile(bExecute := FALSE);
		END_IF


	(* file access complete *)
	E_FILE_DONE:

		bDone := TRUE;
		bBusy := FALSE;

		(* return to IDLE state *)
		eState := E_FILE_IDLE;

END_CASE

END_FUNCTION_BLOCK

// ---- POUs/METS/Common LIB/08_SOFTWARE LIB/File FBs/FB_FILE_Rename.TcPOU
(* rename file *)
FUNCTION_BLOCK FB_FILE_Rename
VAR_INPUT
	bExecute			: BOOL;			(* set TRUE to copy multiple files *)
	strPathSource		: T_MaxString;	(* path of SOURCE folder, can include file name as well if file name is to be changed *)
	strPathTarget		: T_MaxString;	(* path of TARGET folder, can include file name as well if file name is to be changed *)
	strFileName			: T_MaxString;	(* file name to be moved, leave blank if file name is included in paths *)
	tTimeout			: TIME;			(* timeout for each file operation *)
END_VAR
VAR_OUTPUT
	bDone				: BOOL;			(* TRUE = file access complete *)
	bBusy				: BOOL;			(* TRUE = file access in progress *)
	bError				: BOOL;			(* TRUE = error occurred during process *)
	nErrorID			: UDINT;		(* error code *)
END_VAR
VAR
	fbExecute			: R_TRIG;
	eState				: E_FILE_State;
	eErrorState			: E_FILE_State;
	fbDeleteFile		: FB_FileDelete;
	fbMoveFile			: FB_FileRename;
END_VAR
(*
-------------------------------------------------------------------------------------------------
Date		Version	Author	Comments
-------------------------------------------------------------------------------------------------
30/01/2015	3.00.00	PB		Moved from Sewtec_CaseTrace.lib

-------------------------------------------------------------------------------------------------
07/06/2010	1.04.00	PB		Initial release

-------------------------------------------------------------------------------------------------
*)

(* compare files on rising edge of bExecute *)
fbExecute(CLK := bExecute);

CASE eState OF

	(* idle state *)
	E_FILE_IDLE:

		(* start new cycle *)
		IF fbExecute.Q = TRUE THEN

			(* reset outputs *)
			bDone := FALSE;
			bBusy := TRUE;
			bError := FALSE;
			nErrorID := 0;
			eErrorState := eState;

			eState := E_FILE_DELETE;

		(* reset status outputs when no cycle is required and bExecute is reset *)
		ELSIF bExecute = FALSE THEN

			bDone := FALSE;
			bBusy := FALSE;
			bError := FALSE;
			nErrorID := 0;
		END_IF


	(* delete target file *)
	E_FILE_DELETE:

		(* delete file *)
		fbDeleteFile(
			sNetId		:= '',
			sPathName	:= CONCAT(strPathTarget, strFileName),
			ePath		:= PATH_GENERIC,
			bExecute	:= TRUE,
			tTimeout	:= tTimeout
		);

		(* file delete completed *)
		IF fbDeleteFile.bBusy = FALSE THEN

			(* file delete completed OK *)
			IF fbDeleteFile.bError = FALSE THEN

				eState := E_FILE_MOVE;

			(* file delete error *)
			ELSE

				(* file did not exist, OK to move file to TARGET folder *)
				IF fbDeleteFile.nErrId = 1804 THEN

					eState := E_FILE_MOVE;

				(* other file delete error occurred *)
				ELSE

				(* no error has previously occurred *)
					IF bError = FALSE THEN

						(* log error code and failure state *)
						bError := TRUE;
						nErrorID := fbDeleteFile.nErrId;
						eErrorState := eState;
					END_IF

					(* sequence complete *)
					eState := E_FILE_ABORT;
				END_IF
			END_IF

			(* close off fbFileDelete *)
			fbDeleteFile(bExecute := FALSE);
		END_IF


	(* move source file to destination file *)
	E_FILE_MOVE:

		(* move file *)
		fbMoveFile(
			sNetId		:= '',
			sOldName	:= CONCAT(strPathSource, strFileName),
			sNewName	:= CONCAT(strPathTarget, strFileName),
			ePath		:= PATH_GENERIC,
			bExecute	:= TRUE,
			tTimeout	:= tTimeout,
		);
		
		(* file move completed *)
		IF fbMoveFile.bBusy = FALSE THEN

			(* file move completed OK *)
			IF fbMoveFile.bError = FALSE THEN

				eState := E_FILE_DONE;

			(* file move error *)
			ELSE

				(* no error has previously occurred *)
				IF bError = FALSE THEN

					(* log error code and failure state *)
					bError := TRUE;
					nErrorID := fbMoveFile.nErrId;
					eErrorState := eState;
				END_IF

				(* abandon attempt to move file *)
				eState := E_FILE_DONE;
			END_IF

			(* close off fbMoveFile *)
			fbMoveFile(bExecute := FALSE);
		END_IF


	(* file access complete *)
	E_FILE_DONE:

		bDone := TRUE;
		bBusy := FALSE;

		(* return to IDLE state *)
		eState := E_FILE_IDLE;

END_CASE

END_FUNCTION_BLOCK

// ---- POUs/METS/Common LIB/08_SOFTWARE LIB/File FBs/FB_FILE_WriteByByte.TcPOU
(* write data from the source array to the target file in byte form *)
FUNCTION_BLOCK FB_FILE_WriteByByte
VAR_INPUT
	bExecute			: BOOL;			(* set TRUE to write file *)
	pSourceAddr			: POINTER TO BYTE;	(* pointer to array of bytes containing data to be written *)
	nSourceSize			: UDINT;		(* number of bytes to write to file *)
	strPathFile			: T_MaxString;	(* full path\file of output file *)
	tTimeout			: TIME;			(* timeout for each file operation *)
END_VAR
VAR_OUTPUT
	bDone				: BOOL;			(* TRUE = file access complete *)
	bBusy				: BOOL;			(* TRUE = file access in progress *)
	bError				: BOOL;			(* TRUE = error occurred during process *)
	nErrorID			: UDINT;		(* error code *)
	nBytesWritten		: UDINT;		(* number of bytes written to specified file *)
END_VAR
VAR
	eState				: E_FILE_State;
	eErrorState			: E_FILE_State;
	fbExecute			: R_TRIG;
	bReWriteFile		: BOOL;
	fbOpenFile			: FB_FileOpen;
	hFileHandle			: UINT;
	fbWriteFile			: FB_FileWrite;
	fbCloseFile			: FB_FileClose;
	nFileWrites			: BYTE;
END_VAR
(*
-------------------------------------------------------------------------------------------------
Date		Version	Author	Comments
-------------------------------------------------------------------------------------------------
30/01/2015	3.00.00	PB		Moved from Sewtec_CaseTrace.lib

-------------------------------------------------------------------------------------------------
21/03/2012	1.37.04	PB		Number of bytes written by FB_FileWrite now checked against nSourceSize, re-write file if valus is incorrect
							Attempt to write file 3 times before returning error
02/03/2010	1.00.00	PB		Initial release

-------------------------------------------------------------------------------------------------
*)

(* load XML file on rising edge of bExecute *)
fbExecute(CLK := bExecute);

CASE eState OF

	(* idle state *)
	E_FILE_IDLE:

		(* start new cycle *)
		IF fbExecute.Q = TRUE THEN

			(* reset outputs *)
			bDone := FALSE;
			bBusy := TRUE;
			bError := FALSE;
			nErrorID := 0;
			eErrorState := eState;
			bReWriteFile := FALSE;
			nFileWrites := 0;

			eState := E_FILE_OPEN;

		(* reset status outputs when no cycle is required and bExecute is reset *)
		ELSIF bExecute = FALSE THEN

			bDone := FALSE;
			bBusy := FALSE;
			bError := FALSE;
			nErrorID := 0;
		END_IF

	(* open file *)
	E_FILE_OPEN:

		(* open specified file for writing in binary mode *)
		fbOpenFile(
			sNetId		:= '',
			sPathName	:= strPathFile,
			nMode		:= FOPEN_MODEWRITE OR FOPEN_MODEBINARY,
			ePath		:= PATH_GENERIC,
			bExecute	:= TRUE,
			tTimeout	:= t#1s,
			hFile		=> hFileHandle
		);

		(* file open completed *)
		IF fbOpenFile.bBusy = FALSE THEN

			(* file open completed OK *)
			IF fbOpenFile.bError = FALSE THEN

				eState := E_FILE_WRITE;

			(* file open error *)
			ELSE

				(* no previous error has occurred *)
				IF bError = FALSE THEN

					(* log error code and failure state *)
					bError := TRUE;
					nErrorID := fbOpenFile.nErrId;
					eErrorState := eState;
				END_IF

				(* abandon attempt to read file *)
				eState := E_FILE_DONE;
			END_IF

			(* close off fbOpenFile *)
			fbOpenFile(bExecute := FALSE);
		END_IF


	(* write file *)
	E_FILE_WRITE:

		(* write data to open file *)
		fbWriteFile(
			sNetId		:= '',
			hFile		:= hFileHandle,
			pWriteBuff	:= pSourceAddr,
			cbWriteLen	:= nSourceSize,
			bExecute	:= TRUE,
			tTimeout	:= tTimeout,
			cbWrite		=> nBytesWritten
		);

		(* file write completed *)
		IF fbWriteFile.bBusy = FALSE THEN

			(* file write completed OK *)
			IF fbWriteFile.bError = FALSE THEN

				(* number of bytes written was correct *)
				IF nBytesWritten = nSourceSize THEN

					bReWriteFile := FALSE;

				(* number of bytes written was not correct *)
				ELSE

					(* set re-write flag *)
					bReWriteFile := TRUE;
				END_IF

				eState := E_FILE_CLOSE;

			(* file write error *)
			ELSE

				(* no previous error has occurred *)
				IF bError = FALSE THEN

					(* log error code and failure state *)
					bError := TRUE;
					nErrorID := fbWriteFile.nErrId;
					eErrorState := eState;
				END_IF

				(* abandon write and close file *)
				eState := E_FILE_CLOSE;
			END_IF

			(* close off fbReadFile *)
			fbWriteFile(bExecute := FALSE);
		END_IF


	(* close file *)
	E_FILE_CLOSE:

		(* close and release file for future use *)
		fbCloseFile(
			sNetId		:= '',
			hFile		:= hFileHandle,
			bExecute	:= TRUE,
			tTimeout	:= t#1s,
		);

		(* file close completed *)
		IF fbCloseFile.bBusy = FALSE THEN

			(* count number of open-write-close attempts *)
			nFileWrites := nFileWrites + 1;

			(* file close completed OK *)
			IF fbCloseFile.bError = FALSE THEN

				(* file write OK *)
				IF bReWriteFile = FALSE THEN

					eState := E_FILE_DONE;

				(* file write failed *)
				ELSE

					(* 3 write attempts failed *)
					IF nFileWrites >= 3 THEN

						bError := TRUE;
						nErrorID := 16#FFFFFFFF;
						eErrorState := eState;

						eState := E_FILE_DONE;

					(* re-try to write file *)
					ELSE

						eState := E_FILE_OPEN;
					END_IF
				END_IF

			(* file close error *)
			ELSE

				(* no error occurred with FileOpen or FileRead *)
				IF bError = FALSE THEN

					(* log error code and failure state *)
					bError := TRUE;
					nErrorID := fbCloseFile.nErrId;
					eErrorState := eState;
				END_IF

				eState := E_FILE_DONE;
			END_IF

			(* close off fbCloseFile *)
			fbCloseFile(bExecute := FALSE);
		END_IF


	(* file access complete *)
	E_FILE_DONE:

		bDone := TRUE;
		bBusy := FALSE;

		(* return to IDLE state *)
		eState := E_FILE_IDLE;

END_CASE

END_FUNCTION_BLOCK

// ---- POUs/METS/Common LIB/08_SOFTWARE LIB/File FBs/F_FILE_CompareFileTime.TcPOU
(* compare file time for 2 files *)
FUNCTION F_FILE_CompareFileTime : DINT
VAR_INPUT
	nFileTime1		: T_FILETIME;
	nFileTime2		: T_FILETIME;
END_VAR
VAR
	nULarge1		: T_ULARGE_INTEGER;
	nULarge2		: T_ULARGE_INTEGER;
END_VAR
(*
-------------------------------------------------------------------------------------------------
Date		Version	Author	Comments
-------------------------------------------------------------------------------------------------
30/01/2015	3.00.00	PB		Moved from Sewtec_CaseTrace.lib

-------------------------------------------------------------------------------------------------
06/09/2012	1.41.00	PB		Initial release

-------------------------------------------------------------------------------------------------

F_FILE_CompareFileTime > 0		nFileTime1 > nFileTime2
F_FILE_CompareFileTime = 0		nFileTime1 = nFileTime2
F_FILE_CompareFileTime < 0		nFileTime1 < nFileTime2
*)

(* convert T_FILETIME to T_ULARGE_INTEGER *)
MEMMOVE(ADR(nULarge1), ADR(nFileTime1), SIZEOF(nULarge1));
MEMMOVE(ADR(nULarge2), ADR(nFileTime2), SIZEOF(nULarge2));

(* 64-bit compare *)
F_FILE_CompareFileTime := UInt64Cmp64(nULarge1, nULarge2);

END_FUNCTION

// ---- POUs/METS/Common LIB/08_SOFTWARE LIB/File FBs/F_FILE_FileTimeToULarge.TcPOU
(* convert value from 64-bit T_FILETIME to 64-bit T_ULARGE_INTEGER *)
FUNCTION F_FILE_FileTimeToULarge : T_ULARGE_INTEGER
VAR_INPUT
	sFileTime		: T_FILETIME;
END_VAR
VAR
END_VAR
(*
-------------------------------------------------------------------------------------------------
Date		Version	Author	Comments
-------------------------------------------------------------------------------------------------
26/03/2012	1.38.00	PB		Initial release

-------------------------------------------------------------------------------------------------
*)

MEMMOVE(ADR(F_FILE_FileTimeToULarge), ADR(sFileTime), SIZEOF(F_FILE_FileTimeToULarge));

END_FUNCTION

// ---- POUs/METS/Common LIB/08_SOFTWARE LIB/File FBs/F_FILE_SetFileExtension.TcPOU
FUNCTION F_FILE_SetFileExtension : T_MaxString
VAR_INPUT
	Filename 						: T_MaxString;
	Extension 						: T_FileExtension;
END_VAR
VAR
	Result 							: T_MaxString;
	DotPosition						: INT;
END_VAR

IF LEFT(Extension,1) <> cDOT_CHAR THEN (*No leading dot character found, so add it *)
	Extension := CONCAT(cDOT_CHAR, Extension);
END_IF

DotPosition := FIND(Filename, cDOT_CHAR);
IF DotPosition = 0 THEN (*No file extension - append new file extension*)
	Result := CONCAT(Filename,Extension);
ELSE
	Result := CONCAT(LEFT(Filename, DotPosition-1),Extension);
END_IF

F_FILE_SetFileExtension := Result;

END_FUNCTION

// ---- POUs/METS/Common LIB/08_SOFTWARE LIB/File FBs/F_FILE_SplitFilename.TcPOU
FUNCTION F_FILE_SplitFilename : T_MaxString
VAR_INPUT
	strPathFile		: T_MaxString;
END_VAR
VAR
	nMaxIndex		: INT;
	nIndex			: INT;
	strChar			: STRING(1);
END_VAR
(*
-------------------------------------------------------------------------------------------------
Date		Version	Author	Comments
-------------------------------------------------------------------------------------------------
30/01/2015	3.00.00	PB		Moved from Sewtec_CaseTrace.lib

-------------------------------------------------------------------------------------------------
26/03/2012	1.38.00	PB		Initial release

-------------------------------------------------------------------------------------------------
*)

(* total no of chars in string *)
nMaxIndex := LEN(strPathFile);

(* initialise output *)
F_FILE_SplitFilename := '';

(* scan each char in string *)
FOR nIndex := 0 TO nMaxIndex - 1 DO

	(* start from end of string *)
	strChar := MID(strPathFile, 1, nMaxIndex - nIndex);

	(* last '\' char is string separates path and file name *)
	IF strChar = '\' THEN

		F_FILE_SplitFilename := RIGHT(strPathFile, nIndex);
		EXIT;
	END_IF
END_FOR

END_FUNCTION

// ---- POUs/METS/Common LIB/08_SOFTWARE LIB/File FBs/F_FILE_SplitPath.TcPOU
FUNCTION F_FILE_SplitPath : T_MaxString
VAR_INPUT
	strPathFile		: T_MaxString;
END_VAR
VAR
	nMaxIndex		: INT;
	nIndex			: INT;
	strChar			: STRING(1);
END_VAR
(*
-------------------------------------------------------------------------------------------------
Date		Version	Author	Comments
-------------------------------------------------------------------------------------------------
30/01/2015	3.00.00	PB		Moved from Sewtec_CaseTrace.lib

-------------------------------------------------------------------------------------------------
26/03/2012	1.38.00	PB		Initial release

-------------------------------------------------------------------------------------------------
*)

(* total no of chars in string *)
nMaxIndex := LEN(strPathFile);

(* initialise output *)
F_FILE_SplitPath := '';

(* scan each char in string *)
FOR nIndex := 0 TO nMaxIndex - 1 DO

	(* start from end of string *)
	strChar := MID(strPathFile, 1, nMaxIndex - nIndex);

	(* last '\' char is string separates path and file name *)
	IF strChar = '\' THEN

		F_FILE_SplitPath := LEFT(strPathFile, nMaxIndex - nIndex);
		EXIT;
	END_IF
END_FOR

END_FUNCTION

// ---- POUs/METS/Common LIB/08_SOFTWARE LIB/File FBs/F_FILE_TIME_GT.TcPOU
(*
Compares two T_FILETIME structures. Returs true if ftTime1 > ftTime2. i.e ftTime1 is LATER (more recent) than ftTime2.
*)
FUNCTION F_FILE_TIME_GT : BOOL
VAR_INPUT
	ftTime1			: T_FILETIME;
	ftTime2			: T_FILETIME;
END_VAR
VAR
END_VAR

IF ftTime1.dwHighDateTime > ftTime2.dwHighDateTime THEN
	F_FILE_TIME_GT := TRUE;
	RETURN;
ELSIF ftTime1.dwHighDateTime = ftTime2.dwHighDateTime AND ftTime1.dwLowDateTime >ftTime2.dwLowDateTime  THEN
	F_FILE_TIME_GT := TRUE;
	RETURN;
ELSE
	F_FILE_TIME_GT := FALSE;
END_IF

END_FUNCTION

// ---- POUs/METS/Common LIB/08_SOFTWARE LIB/File FBs/F_FILE_ULargeToFileTime.TcPOU
(* convert value from 64-bit T_ULARGE_INTEGER to 64-bit T_FILETIME *)
FUNCTION F_FILE_ULargeToFileTime : T_FILETIME
VAR_INPUT
	nULarge		: T_ULARGE_INTEGER;
END_VAR
VAR
END_VAR
(*
-------------------------------------------------------------------------------------------------
Date		Version	Author	Comments
-------------------------------------------------------------------------------------------------
03/08/2012	1.39.00	PB		Initial release

-------------------------------------------------------------------------------------------------
*)

MEMMOVE(ADR(F_FILE_ULargeToFileTime), ADR(nULarge), SIZEOF(nULarge));

END_FUNCTION

// ---- POUs/METS/Common LIB/08_SOFTWARE LIB/IP Address FBs/F_IP_AddressPort.TcPOU
(* determine if IP address and Port have been configured *)
FUNCTION F_IP_AddressPort : BOOL
VAR_INPUT
	strIPAddress	: T_IPv4Addr;
	nPort			: UINT;
END_VAR
VAR
END_VAR
(*
-------------------------------------------------------------------------------------------------
Date		Version	Author	Comments
-------------------------------------------------------------------------------------------------
30/01/2015	3.00.00	PB		Initial release

-------------------------------------------------------------------------------------------------
*)

(* '0.0.0.0' indicates blank or invalid IP address in strIPAddress, nPort must not be 0 *)
IF F_CreateIPv4Addr(F_ScanIPv4AddrIds(strIPAddress)) <> '0.0.0.0' AND nPort > 0 THEN

	(* valid *)
	F_IP_AddressPort := TRUE;

(* IP address or Port not set *)
ELSE

	F_IP_AddressPort := FALSE;
END_IF

END_FUNCTION

// ---- POUs/METS/Common LIB/08_SOFTWARE LIB/Logger FBs/FB_LOG_FileWriteError.TcPOU
FUNCTION_BLOCK FB_LOG_FileWriteError
VAR_INPUT
	bLogData					: BOOL;
	nWriteErrorID				: UDINT;
	stCTDateTime				: ST_SYSTEM_DateTime;
	strFileName					: T_MaxString;
END_VAR
VAR_IN_OUT
	aLogFileWriteError			: ARRAY[1..10] OF ST_LOG_FileWriteError;
END_VAR
VAR_OUTPUT
	bDone					: BOOL;
END_VAR
VAR
	rtExecute					: R_TRIG;
	sTimeStamp				: STRING;
END_VAR

rtExecute(CLK:=bLogData);

IF rtExecute.Q THEN
	MEMMOVE(ADR(aLogFileWriteError[2]), ADR(aLogFileWriteError[1]), SIZEOF(aLogFileWriteError) - SIZEOF(aLogFileWriteError[1]));


	aLogFileWriteError[1].nWriteErrorID := nWriteErrorID;
	aLogFileWriteError[1].strFileName := strFileName;
	aLogFileWriteError[1].sTimeStamp := F_SYSTEM_SystemTimeAsISO8601(stCTDateTime.sSystemTime, stCTDateTime.sUTCTimeZoneOffset);
	bDone	:= TRUE;

